# B&R Automation Studio project CControl_Gschneitner
Automation Studio 4.12.9.18 SP; technology packages: mapp 5.24.6

## Configuration 2_07

CPU 4PPC30.0702-21B, AutomationRuntime S4.93, Build 4.1.2, Safety 0.0, Vc V4.73.5

### Task classes (Cpu.sw)
```
Cyclic#1 (cycle 10000 us, tolerance 10000 us):
  eUhr <- Util.eUhr.prg
  UsbLink <- CSV.UsbLink.prg
Cyclic#2 (cycle 20000 us, tolerance 20000 us):
  hmiMain <- Visualisierung.hmiMain.prg
  System <- Util.System.prg
  StartStopp <- Steuerung.StartStopp.prg
  mappPara <- Util.mappPara.prg
Cyclic#3 (cycle 50000 us, tolerance 50000 us):
  io207 <- IO.io207.prg
  aktorenMap <- IO.aktorenMapping.prg
  boxenMappi <- IO.boxenMapping.prg
  Ablaufstrg <- Ablaufsteuerung.Ablaufstrg.prg
  Leistung <- Regelung.Leistung.prg
  Sitemanage <- Sitemanager.Sitemanager.prg
Cyclic#4 (cycle 100000 us, tolerance 100000 us):
  Nutzung <- Util.Nutzung.prg
  Alarm <- Alarmsystem.Alarm.prg
  Berechnung <- Berechnung.Berechnung.prg
Cyclic#5 (cycle 200000 us, tolerance 200000 us):
  Energiemes <- IO.Energiemessung.prg
  hmiConnect <- Visualisierung.hmiConnect.prg
Cyclic#6 (cycle 500000 us, tolerance 500000 us):
  CSV01_EXT <- CSV.CSV01_EXT.prg
  CSV01_PRG <- CSV.CSV01_PRG.prg
DataObjects: CSV01_CFG <- CSV.CSV01_CFG.dob
VcDataObjects: Visu <- Visualisierung.Visu.dob
Binaries: vccddbox, vccbtn, vcpdvnc, arialbd, vcmgr, vctcal, vcgclass, vcfile, vccnum, TCData, vcfntttf, vcpkat, vcdsloc, vcbclass, udbdef, FWRules, vcpd335x, vccstr, vccalarm, visvc, arial, Visu03, vccshape, vcalarm, vcpfppct, Visu01, vccdt, vcptelo, vcchspot, vcpk, vccbmp, vccpopup, vcshared, vcrt, vcnet, Visu02, vcctext, vcctrend, arsvcreg, vcclbox, vccbar, vcdsint, vcpdsw, vccovl, vccline, Config, sysconf, Role, User, ashwd, ashwac, iomap, arconfig, asfw
Libraries: operator, runtime, astime, AsIecCon, standard, sys_lib, AsBrStr, LascoMath, LascoReg, LascoTrock, LascoUtil, LaEntfV2, LascoBoxen, LoopConR, brsystem, asstring, FileIO, DataObj, AsARCfg, visapi, AsUSB, dvframe, IecCheck, MpBase, AsTCP, MpFile, MpRecipe, CControl, CSV, vcresman
```

### Hardware
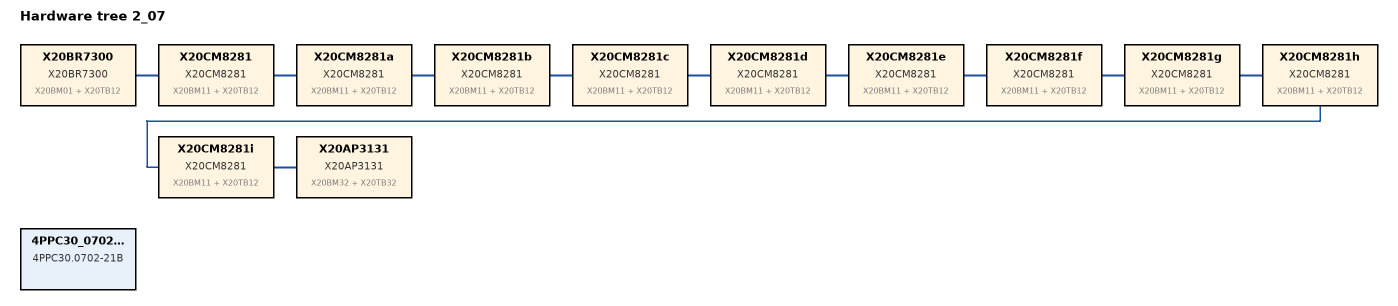
```
4PPC30_0702_21B : 4PPC30.0702-21B v1.1.4.0
  Connector IF3:
    ActivateDevice = 1
    Mode = Manual
    InternetAddress = 10.0.0.2
    SubnetMask = 255.255.255.0
    Vnc1
    VncVcObjectName1 = Visu
    VncKeyMappingFile1 = VC\PS2-Keyboard.dis
    VncMaxConnections1 = 5
    VncRefreshRate1 = 100
  Connector IF4:
    TerminatingResistor = 1
  ConfigurationID = CControl_2_07
  UserPartitionSize = 300
  RemanentGlobalPvSize = 7200
  EnableUsbRemoteInstall = 1
  TimerDeviceType = SWIOTIMER
  Cyclic1Duration = 10000
  Cyclic1Tolerance = 10000
  Cyclic2Duration = 20000
  Cyclic2Tolerance = 20000
  Cyclic3Duration = 50000
  Cyclic3Tolerance = 50000
  Cyclic4Duration = 100000
  Cyclic4Tolerance = 100000
  Cyclic5Duration = 200000
  Cyclic5Tolerance = 200000
  Cyclic6Duration = 500000
  Cyclic6Tolerance = 500000
  Cyclic7Duration = 1000000
  Cyclic7Tolerance = 1000000
  Cyclic8Duration = 10000
  Cyclic8Tolerance = 30000000
  FileDevice1
  FileDeviceName1 = CF
  FileDevicePath1 = F:\
  TimeZone = 140
  ActivateDaylightSavingTime = 1
  FtpUser1
  FtpUsername1 = lasco
  FtpUserPassword1 = KKiL+oKJhPTyxG5QFdiy6FHyy8yLLXpJAQupzJScLRk=
  FtpUserSalt1 = MRssQ874
  FTPAccessRight1 = 0
  FTPdevice1 = ALL
  VcObjectName = Visu
  KeyMappingFile = VC\4PPC30_0702_21B.dis
X20AP3131 : X20AP3131 v1.5.0.0  [SS1 -> X20TB32.SS; SL -> X20BM32.SL1]
  FunctionModel = CANIOBusController
  Supervision = off
  CurrentRatioA = 50
  CurrentRatioB = 50
  CurrentRatioC = 50
X20BM01 : X20BM01 v2.2.0.0
X20BM11 : X20BM11 v1.1.0.0  [X2X1 -> X20BM01.IF1]
X20BM11a : X20BM11 v1.1.0.0  [X2X1 -> X20BM11.X2X2]
X20BM11b : X20BM11 v1.1.0.0  [X2X1 -> X20BM11a.X2X2]
X20BM11c : X20BM11 v1.1.0.0  [X2X1 -> X20BM11b.X2X2]
X20BM11d : X20BM11 v1.1.0.0  [X2X1 -> X20BM11c.X2X2]
X20BM11e : X20BM11 v1.1.0.0  [X2X1 -> X20BM11d.X2X2]
X20BM11f : X20BM11 v1.1.0.0  [X2X1 -> X20BM11e.X2X2]
X20BM11g : X20BM11 v1.1.0.0  [X2X1 -> X20BM11f.X2X2]
X20BM11h : X20BM11 v1.1.0.0  [X2X1 -> X20BM11g.X2X2]
X20BM11i : X20BM11 v1.1.0.0  [X2X1 -> X20BM11h.X2X2]
X20BM32 : X20BM32 v1.1.0.0  [X2X1 -> X20BM11i.X2X2]
X20BR7300 : X20BR7300 v1.7.0.0  [CAN1 -> 4PPC30_0702_21B.IF4; SL -> X20BM01.SL1; SS1 -> X20TB12.SS]
  Supervision = off
X20CM8281 : X20CM8281 v1.4.0.0  [SS1 -> X20TB12a.SS; SL -> X20BM11.SL1]
  FunctionModel = CANIOBusController
  Supervision = off
  ChannelType01AI = 4 to 20mA
  LowerLimitAI = 0
  ChannelType01AO = 0 to 20mA
X20CM8281a : X20CM8281 v1.4.0.0  [SS1 -> X20TB12b.SS; SL -> X20BM11a.SL1]
  FunctionModel = CANIOBusController
  Supervision = off
  ChannelType01AI = 4 to 20mA
  LowerLimitAI = 0
  ChannelType01AO = 0 to 20mA
X20CM8281b : X20CM8281 v1.4.0.0  [SS1 -> X20TB12c.SS; SL -> X20BM11b.SL1]
  FunctionModel = CANIOBusController
  Supervision = off
  ChannelType01AI = 4 to 20mA
  LowerLimitAI = 0
  ChannelType01AO = 0 to 20mA
X20CM8281c : X20CM8281 v1.4.0.0  [SS1 -> X20TB12d.SS; SL -> X20BM11c.SL1]
  FunctionModel = CANIOBusController
  Supervision = off
  ChannelType01AI = 4 to 20mA
  LowerLimitAI = 0
X20CM8281d : X20CM8281 v1.4.0.0  [SS1 -> X20TB12e.SS; SL -> X20BM11d.SL1]
  FunctionModel = CANIOBusController
  Supervision = off
  ChannelType01AI = 4 to 20mA
  LowerLimitAI = 0
X20CM8281e : X20CM8281 v1.4.0.0  [SS1 -> X20TB12f.SS; SL -> X20BM11e.SL1]
  FunctionModel = CANIOBusController
  Supervision = off
  ChannelType01AI = 4 to 20mA
  LowerLimitAI = 0
X20CM8281f : X20CM8281 v1.4.0.0  [SS1 -> X20TB12g.SS; SL -> X20BM11f.SL1]
  FunctionModel = CANIOBusController
  Supervision = off
  ChannelType01AI = 4 to 20mA
  LowerLimitAI = 0
  ChannelType01AO = 0 to 20mA
X20CM8281g : X20CM8281 v1.4.0.0  [SS1 -> X20TB12h.SS; SL -> X20BM11g.SL1]
  FunctionModel = CANIOBusController
  Supervision = off
  ChannelType01AI = 4 to 20mA
  LowerLimitAI = 0
X20CM8281h : X20CM8281 v1.4.0.0  [SS1 -> X20TB12i.SS; SL -> X20BM11h.SL1]
  FunctionModel = CANIOBusController
  Supervision = off
X20CM8281i : X20CM8281 v1.4.0.0  [SS1 -> X20TB12j.SS; SL -> X20BM11i.SL1]
  FunctionModel = CANIOBusController
  Supervision = off
  ChannelType01AI = 4 to 20mA
X20TB12 : X20TB12 v1.0.0.0
X20TB12a : X20TB12 v1.0.0.0
X20TB12b : X20TB12 v1.0.0.0
X20TB12c : X20TB12 v1.0.0.0
X20TB12d : X20TB12 v1.0.0.0
X20TB12e : X20TB12 v1.0.0.0
X20TB12f : X20TB12 v1.0.0.0
X20TB12g : X20TB12 v1.0.0.0
X20TB12h : X20TB12 v1.0.0.0
X20TB12i : X20TB12 v1.0.0.0
X20TB12j : X20TB12 v1.0.0.0
X20TB32 : X20TB32 v1.0.0.1
```

### IoMap.iom - 4PPC30_0702_21B/IoMap.iom
```iecst
VAR_CONFIG
	::io207:brModul01.ModulOk AT %IX."X20BR7300".IF1.ST1.ModuleOk;
	::io207:cmModul02.ModulOk AT %IX."X20CM8281".ModuleOk;
	::io207:cmModul02.di01 AT %IX."X20CM8281".DigitalInput01;
	::io207:cmModul02.di02  AT %IX."X20CM8281".DigitalInput02;
	::io207:cmModul02.di03 AT %IX."X20CM8281".DigitalInput03;
	::io207:cmModul02.di04  AT %IX."X20CM8281".DigitalInput04;
	::io207:cmModul02.do01 AT %QX."X20CM8281".DigitalOutput01;
	::io207:cmModul02.do02 AT %QX."X20CM8281".DigitalOutput02;
	::io207:cmModul02.ai01 AT %IW."X20CM8281".AnalogInput01;
	::io207:cmModul02.ao01 AT %QW."X20CM8281".AnalogOutput01;
	::io207:cmModul02.StatusInput01 AT %IB."X20CM8281".StatusInput01;
	::io207:cmModul03.ModulOk AT %IX."X20CM8281a".ModuleOk;
	::io207:cmModul03.di01 AT %IX."X20CM8281a".DigitalInput01;
	::io207:cmModul03.di02  AT %IX."X20CM8281a".DigitalInput02;
	::io207:cmModul03.di03  AT %IX."X20CM8281a".DigitalInput03;
	::io207:cmModul03.di04  AT %IX."X20CM8281a".DigitalInput04;
	::io207:cmModul03.do01 AT %QX."X20CM8281a".DigitalOutput01;
	::io207:cmModul03.do02 AT %QX."X20CM8281a".DigitalOutput02;
	::io207:cmModul03.ai01 AT %IW."X20CM8281a".AnalogInput01;
	::io207:cmModul03.ao01 AT %QW."X20CM8281a".AnalogOutput01;
	::io207:cmModul03.StatusInput01 AT %IB."X20CM8281a".StatusInput01;
	::io207:cmModul04.ModulOk AT %IX."X20CM8281b".ModuleOk;
	::io207:cmModul04.di01 AT %IX."X20CM8281b".DigitalInput01;
	::io207:cmModul04.di02 AT %IX."X20CM8281b".DigitalInput02;
	::io207:cmModul04.di03 AT %IX."X20CM8281b".DigitalInput03;
	::io207:cmModul04.di04 AT %IX."X20CM8281b".DigitalInput04;
	::io207:cmModul04.do01 AT %QX."X20CM8281b".DigitalOutput01;
	::io207:cmModul04.do02 AT %QX."X20CM8281b".DigitalOutput02;
	::io207:cmModul04.ai01 AT %IW."X20CM8281b".AnalogInput01;
	::io207:cmModul04.ao01 AT %QW."X20CM8281b".AnalogOutput01;
	::io207:cmModul04.StatusInput01 AT %IB."X20CM8281b".StatusInput01;
	::io207:cmModul05.ModulOk AT %IX."X20CM8281c".ModuleOk;
	::io207:cmModul05.di01 AT %IX."X20CM8281c".DigitalInput01;
	::io207:cmModul05.di02 AT %IX."X20CM8281c".DigitalInput02;
	::io207:cmModul05.di03 AT %IX."X20CM8281c".DigitalInput03;
	::io207:cmModul05.di04 AT %IX."X20CM8281c".DigitalInput04;
	::io207:cmModul05.do01 AT %QX."X20CM8281c".DigitalOutput01;
	::io207:cmModul05.do02 AT %QX."X20CM8281c".DigitalOutput02;
	::io207:cmModul05.ai01 AT %IW."X20CM8281c".AnalogInput01;
	::io207:cmModul05.ao01 AT %QW."X20CM8281c".AnalogOutput01;
	::io207:cmModul05.StatusInput01 AT %IB."X20CM8281c".StatusInput01;
	::io207:cmModul06.ModulOk AT %IX."X20CM8281d".ModuleOk;
	::io207:cmModul06.di01 AT %IX."X20CM8281d".DigitalInput01;
	::io207:cmModul06.di02 AT %IX."X20CM8281d".DigitalInput02;
	::io207:cmModul06.di03 AT %IX."X20CM8281d".DigitalInput03;
	::io207:cmModul06.di04 AT %IX."X20CM8281d".DigitalInput04;
	::io207:cmModul06.do01 AT %QX."X20CM8281d".DigitalOutput01;
	::io207:cmModul06.do02 AT %QX."X20CM8281d".DigitalOutput02;
	::io207:cmModul06.ai01 AT %IW."X20CM8281d".AnalogInput01;
	::io207:cmModul06.ao01 AT %QW."X20CM8281d".AnalogOutput01;
	::io207:cmModul06.StatusInput01 AT %IB."X20CM8281d".StatusInput01;
	::io207:cmModul07.ModulOk AT %IX."X20CM8281e".ModuleOk;
	::io207:cmModul07.di01 AT %IX."X20CM8281e".DigitalInput01;
	::io207:cmModul07.di02 AT %IX."X20CM8281e".DigitalInput02;
	::io207:cmModul07.di03 AT %IX."X20CM8281e".DigitalInput03;
	::io207:cmModul07.di04 AT %IX."X20CM8281e".DigitalInput04;
	::io207:cmModul07.do01 AT %QX."X20CM8281e".DigitalOutput01;
	::io207:cmModul07.do02 AT %QX."X20CM8281e".DigitalOutput02;
	::io207:cmModul07.ai01 AT %IW."X20CM8281e".AnalogInput01;
	::io207:cmModul07.ao01 AT %QW."X20CM8281e".AnalogOutput01;
	::io207:cmModul07.StatusInput01 AT %IB."X20CM8281e".StatusInput01;
	::io207:cmModul08.ModulOk AT %IX."X20CM8281f".ModuleOk;
	::io207:cmModul08.di01 AT %IX."X20CM8281f".DigitalInput01;
	::io207:cmModul08.di02 AT %IX."X20CM8281f".DigitalInput02;
	::io207:cmModul08.di03 AT %IX."X20CM8281f".DigitalInput03;
	::io207:cmModul08.di04 AT %IX."X20CM8281f".DigitalInput04;
	::io207:cmModul08.do01 AT %QX."X20CM8281f".DigitalOutput01;
	::io207:cmModul08.do02 AT %QX."X20CM8281f".DigitalOutput02;
	::io207:cmModul08.ai01 AT %IW."X20CM8281f".AnalogInput01;
	::io207:cmModul08.ao01 AT %QW."X20CM8281f".AnalogOutput01;
	::io207:cmModul08.StatusInput01 AT %IB."X20CM8281f".StatusInput01;
	::io207:cmModul09.ModulOk AT %IX."X20CM8281g".ModuleOk;
	::io207:cmModul09.di01 AT %IX."X20CM8281g".DigitalInput01;
	::io207:cmModul09.di02 AT %IX."X20CM8281g".DigitalInput02;
	::io207:cmModul09.di03 AT %IX."X20CM8281g".DigitalInput03;
	::io207:cmModul09.di04 AT %IX."X20CM8281g".DigitalInput04;
	::io207:cmModul09.do01 AT %QX."X20CM8281g".DigitalOutput01;
	::io207:cmModul09.do02 AT %QX."X20CM8281g".DigitalOutput02;
	::io207:cmModul09.ai01 AT %IW."X20CM8281g".AnalogInput01;
	::io207:cmModul09.ao01 AT %QW."X20CM8281g".AnalogOutput01;
	::io207:cmModul09.StatusInput01 AT %IB."X20CM8281g".StatusInput01;
	::io207:cmModul10.ModulOk AT %IX."X20CM8281h".ModuleOk;
	::io207:cmModul10.di01 AT %IX."X20CM8281h".DigitalInput01;
	::io207:cmModul10.di02 AT %IX."X20CM8281h".DigitalInput02;
	::io207:cmModul10.di03 AT %IX."X20CM8281h".DigitalInput03;
	::io207:cmModul10.di04 AT %IX."X20CM8281h".DigitalInput04;
	::io207:cmModul10.do01 AT %QX."X20CM8281h".DigitalOutput01;
	::io207:cmModul10.do02 AT %QX."X20CM8281h".DigitalOutput02;
	::io207:cmModul10.ai01 AT %IW."X20CM8281h".AnalogInput01;
	::io207:cmModul10.ao01 AT %QW."X20CM8281h".AnalogOutput01;
	::io207:cmModul10.StatusInput01 AT %IB."X20CM8281h".StatusInput01;
	::io207:cmModul11.ModulOk AT %IX."X20CM8281i".ModuleOk;
	::io207:cmModul11.di01 AT %IX."X20CM8281i".DigitalInput01;
	::io207:cmModul11.di02 AT %IX."X20CM8281i".DigitalInput02;
	::io207:cmModul11.di03 AT %IX."X20CM8281i".DigitalInput03;
	::io207:cmModul11.di04 AT %IX."X20CM8281i".DigitalInput04;
	::io207:cmModul11.do01 AT %QX."X20CM8281i".DigitalOutput01;
	::io207:cmModul11.do02 AT %QX."X20CM8281i".DigitalOutput02;
	::io207:cmModul11.ai01 AT %IW."X20CM8281i".AnalogInput01;
	::io207:cmModul11.ao01 AT %QW."X20CM8281i".AnalogOutput01;
	::io207:cmModul11.StatusInput01 AT %IB."X20CM8281i".StatusInput01;
	::Energiemes:apModulEnergie.ModulOk AT %IX."X20AP3131".ModuleOk;
	::Energiemes:apModulEnergie.PmeanT AT %IW."X20AP3131".PmeanT;
	::Energiemes:apModulEnergie.QmeanT AT %IW."X20AP3131".QmeanT;
	::Energiemes:apModulEnergie.SmeanT AT %IW."X20AP3131".SmeanT;
	::Energiemes:apModulEnergie.PFmeanT AT %IW."X20AP3131".PFmeanT;
	::Energiemes:apModulEnergie.AenergyT AT %ID."X20AP3131".AenergyT;
	::Energiemes:apModulEnergie.RenergyT AT %ID."X20AP3131".RenergyT;
	::Energiemes:apModulEnergie.SAenergyT AT %ID."X20AP3131".SAenergyT;
	::Energiemes:apModulEnergie.RBClearEnergy AT %IX."X20AP3131".RBClearEnergy;
	::Energiemes:apModulEnergie.TrigDFT AT %QX."X20AP3131".TrigDFT;
	::Energiemes:apModulEnergie.EnabEnergy AT %QX."X20AP3131".EnabEnergy;
	::Energiemes:apModulEnergie.ClearEnergy AT %QX."X20AP3131".ClearEnergy;
	::Energiemes:apModulEnergie.ForceEnergy AT %QX."X20AP3131".ForceEnergy;
END_VAR
```

- Physical/2_07/4PPC30_0702_21B/PvMap.vvm: same as Physical/2_07/4PPC30_0702_21B/Cpu.per
### Config.mprecipexml - 4PPC30_0702_21B/mappServices/Config.mprecipexml
```
Element gMappRecipeLink (Type=mprecipexml)
```

## Configuration 3_04_Plus

CPU 4PPC30.043F-21B, AutomationRuntime S4.93, Build 4.1.2, Safety 0.0, Vc V4.73.5

### Task classes (Cpu.sw)
```
Cyclic#1 (cycle 10000 us, tolerance 10000 us):
  eUhr <- Util.eUhr.prg
  UsbLink <- CSV.UsbLink.prg
Cyclic#2 (cycle 20000 us, tolerance 20000 us):
  hmiMain <- Visualisierung.hmiMain.prg
  System <- Util.System.prg
  StartStopp <- Steuerung.StartStopp.prg
  mappPara <- Util.mappPara.prg
Cyclic#3 (cycle 50000 us, tolerance 50000 us):
  io304 <- IO.io304.prg  // IO-Konfiguration 3.04
  aktorenMap <- IO.aktorenMapping.prg
  boxenMappi <- IO.boxenMapping.prg
  Ablaufstrg <- Ablaufsteuerung.Ablaufstrg.prg
  Leistung <- Regelung.Leistung.prg
  Sitemanage <- Sitemanager.Sitemanager.prg
Cyclic#4 (cycle 100000 us, tolerance 100000 us):
  Nutzung <- Util.Nutzung.prg
  Berechnung <- Berechnung.Berechnung.prg
  Alarm <- Alarmsystem.Alarm.prg
Cyclic#5 (cycle 200000 us, tolerance 200000 us):
  hmiConnect <- Visualisierung.hmiConnect.prg
  Energiemes <- IO.Energiemessung.prg
Cyclic#6 (cycle 500000 us, tolerance 500000 us):
  CSV01_EXT <- CSV.CSV01_EXT.prg
  CSV01_PRG <- CSV.CSV01_PRG.prg
DataObjects: CSV01_CFG <- CSV.CSV01_CFG.dob
VcDataObjects: Visu4Z <- Visualisierung.Visu4Z.dob
Binaries: vccalarm, Visu4Z03, udbdef, vcrt, vccbar, vctcal, visvc, vccpopup, vcfile, vcgclass, vccstr, vcpdsw, vccshape, arial, vccbmp, vcmgr, vcshared, vcctrend, vcchspot, vcdsloc, Visu4Z01, vcctext, vccovl, vcfntttf, arialbd, vcpd335x, vccddbox, vcalarm, vcptelo, vccdt, vccline, vccbtn, Visu4Z02, vcbclass, vcdsint, vcpfppct, TCData, vcclbox, FWRules, vcpk, vccnum, arsvcreg, vcpdvnc, vcpkat, vcnet, sysconf, iomap, asfw, Role, ashwac, ashwd, User, arconfig, Config
Libraries: operator, runtime, astime, AsIecCon, standard, sys_lib, AsBrStr, LascoMath, LascoReg, LascoTrock, LascoUtil, LaEntfV2, LascoBoxen, LoopConR, brsystem, asstring, FileIO, DataObj, AsARCfg, visapi, AsUSB, dvframe, IecCheck, AsTCP, MpRecipe, MpBase, MpFile, CSV, CControl, vcresman
```

### Hardware
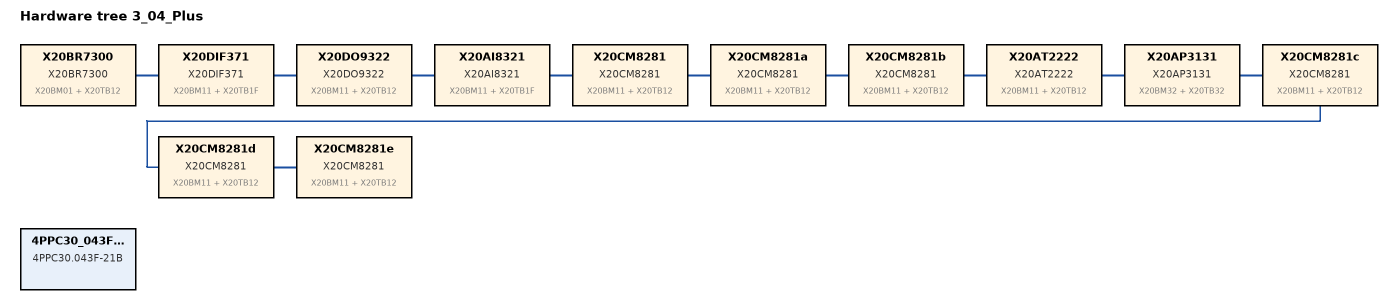
```
4PPC30_043F_21B : 4PPC30.043F-21B v1.1.3.0
  Connector IF3:
    ActivateDevice = 1
    Mode = Manual
    InternetAddress = 10.0.0.2
    SubnetMask = 255.255.255.0
    Vnc1
    VncVcObjectName1 = Visu4Z
    VncKeyMappingFile1 = VC\PS2-Keyboard.dis
    VncMaxConnections1 = 5
    VncRefreshRate1 = 100
  Connector IF4:
    TerminatingResistor = 1
  ConfigurationID = CControl304Plus
  UserPartitionSize = 200
  RemanentGlobalPvSize = 6000
  EnableUsbRemoteInstall = 1
  TimerDeviceType = SWIOTIMER
  Cyclic1Duration = 10000
  Cyclic1Tolerance = 10000
  Cyclic2Duration = 20000
  Cyclic2Tolerance = 20000
  Cyclic3Duration = 50000
  Cyclic3Tolerance = 50000
  Cyclic4Duration = 100000
  Cyclic4Tolerance = 100000
  Cyclic5Duration = 200000
  Cyclic5Tolerance = 200000
  Cyclic6Duration = 500000
  Cyclic6Tolerance = 500000
  Cyclic7Duration = 1000000
  Cyclic7Tolerance = 1000000
  Cyclic8Duration = 10000
  Cyclic8Tolerance = 30000000
  FileDevice1
  FileDeviceName1 = CF
  FileDevicePath1 = F:\
  FtpUser1
  FtpUsername1 = lasco
  FtpUserPassword1 = 97rNj208LBZIZPKyFvn5oul1tIa2LCmp2VBMYd1vER8=
  FtpUserSalt1 = M2zU6OPl
  FTPAccessRight1 = 0
  FTPdevice1 = ALL
  VcObjectName = Visu4Z
  RotationAngle = 180
  KeyMappingFile = VC\4PPC30_043F_21B.dis
X20AI8321 : X20AI8321 v1.5.0.0  [SS1 -> X20TB1F1.SS; SL -> X20BM11b.SL1]
  FunctionModel = CANIOBusController
  Supervision = off
  LowerLimit = 0
  ChannelType01 = 4 to 20mA
  ChannelType02 = 4 to 20mA
  ChannelType03 = 4 to 20mA
  ChannelType04 = 4 to 20mA
  ChannelType05 = 4 to 20mA
  ChannelType06 = 4 to 20mA
  ChannelType07 = 4 to 20mA
  ChannelType08 = 4 to 20mA
X20AP3131 : X20AP3131 v1.5.0.0  [SS1 -> X20TB32.SS; SL -> X20BM32.SL1]
  FunctionModel = CANIOBusController
  Supervision = off
  CurrentRatioA = 50
  CurrentRatioB = 50
  CurrentRatioC = 50
X20AT2222 : X20AT2222 v1.4.0.0  [SS1 -> X20TB12h.SS; SL -> X20BM11i.SL1]
  FunctionModel = CANIOBusController
  Supervision = off
X20BM01 : X20BM01 v2.2.0.0
X20BM11 : X20BM11 v1.1.0.0  [X2X1 -> X20BM01.IF1]
X20BM11a : X20BM11 v1.1.0.0  [X2X1 -> X20BM11.X2X2]
X20BM11b : X20BM11 v1.1.0.0  [X2X1 -> X20BM11a.X2X2]
X20BM11c : X20BM11 v1.1.0.0  [X2X1 -> X20BM11b.X2X2]
X20BM11d : X20BM11 v1.1.0.0  [X2X1 -> X20BM11c.X2X2]
X20BM11e : X20BM11 v1.1.0.0  [X2X1 -> X20BM11d.X2X2]
X20BM11f : X20BM11 v1.1.0.0  [X2X1 -> X20BM32.X2X2]
X20BM11g : X20BM11 v1.1.0.0  [X2X1 -> X20BM11f.X2X2]
X20BM11h : X20BM11 v1.1.0.0  [X2X1 -> X20BM11g.X2X2]
X20BM11i : X20BM11 v1.1.0.0  [X2X1 -> X20BM11e.X2X2]
X20BM32 : X20BM32 v1.1.0.0  [X2X1 -> X20BM11i.X2X2]
X20BR7300 : X20BR7300 v1.7.0.0  [CAN1 -> 4PPC30_043F_21B.IF4; SL -> X20BM01.SL1; SS1 -> X20TB12.SS]
  Supervision = off
X20CM8281 : X20CM8281 v1.4.0.0  [SS1 -> X20TB12b.SS; SL -> X20BM11c.SL1]
  FunctionModel = CANIOBusController
  Supervision = off
  ChannelType01AO = 0 to 20mA
X20CM8281a : X20CM8281 v1.4.0.0  [SS1 -> X20TB12c.SS; SL -> X20BM11d.SL1]
  FunctionModel = CANIOBusController
  Supervision = off
  ChannelType01AI = 4 to 20mA
  LowerLimitAI = 0
  ChannelType01AO = 0 to 20mA
X20CM8281b : X20CM8281 v1.4.0.0  [SS1 -> X20TB12d.SS; SL -> X20BM11e.SL1]
  FunctionModel = CANIOBusController
  Supervision = off
  ChannelType01AI = 4 to 20mA
  LowerLimitAI = 0
X20CM8281c : X20CM8281 v1.4.0.0  [SS1 -> X20TB12e.SS; SL -> X20BM11f.SL1]
  FunctionModel = CANIOBusController
  Supervision = off
  ChannelType01AI = 4 to 20mA
  LowerLimitAI = 0
  ChannelType01AO = 0 to 20mA
X20CM8281d : X20CM8281 v1.4.0.0  [SS1 -> X20TB12f.SS; SL -> X20BM11g.SL1]
  FunctionModel = CANIOBusController
  Supervision = off
  ChannelType01AI = 4 to 20mA
  LowerLimitAI = 0
  ChannelType01AO = 0 to 20mA
X20CM8281e : X20CM8281 v1.4.0.0  [SS1 -> X20TB12g.SS; SL -> X20BM11h.SL1]
  FunctionModel = CANIOBusController
  Supervision = off
  ChannelType01AI = 4 to 20mA
X20DIF371 : X20DIF371 v1.3.0.0  [SS1 -> X20TB1F.SS; SL -> X20BM11.SL1]
  FunctionModel = CANIOBusController
  Supervision = off
X20DO9322 : X20DO9322 v1.7.0.0  [SS1 -> X20TB12a.SS; SL -> X20BM11a.SL1]
  FunctionModel = CANIOBusController
  Supervision = off
X20TB12 : X20TB12 v1.0.0.0
X20TB12a : X20TB12 v1.0.0.0
X20TB12b : X20TB12 v1.0.0.0
X20TB12c : X20TB12 v1.0.0.0
X20TB12d : X20TB12 v1.0.0.0
X20TB12e : X20TB12 v1.0.0.0
X20TB12f : X20TB12 v1.0.0.0
X20TB12g : X20TB12 v1.0.0.0
X20TB12h : X20TB12 v1.0.0.0
X20TB1F : X20TB1F v1.0.0.0
X20TB1F1 : X20TB1F v1.0.0.0
X20TB32 : X20TB32 v1.0.0.1
```

- Physical/3_04_Plus/4PPC30_043F_21B/Cpu.per: same as Physical/2_07/4PPC30_0702_21B/Cpu.per
### IoMap.iom - 4PPC30_043F_21B/IoMap.iom
```iecst
VAR_CONFIG
	::io304:brModul01.ModulOk AT %IX."X20BR7300".IF1.ST1.ModuleOk;
	::io304:diModul02.ModulOk AT %IX."X20DIF371".ModuleOk;
	::io304:diModul02.di01 AT %IX."X20DIF371".DigitalInput01;
	::io304:diModul02.di02 AT %IX."X20DIF371".DigitalInput02;
	::io304:diModul02.di03 AT %IX."X20DIF371".DigitalInput03;
	::io304:diModul02.di04 AT %IX."X20DIF371".DigitalInput04;
	::io304:diModul02.di05 AT %IX."X20DIF371".DigitalInput05;
	::io304:diModul02.di06 AT %IX."X20DIF371".DigitalInput06;
	::io304:diModul02.di07 AT %IX."X20DIF371".DigitalInput07;
	::io304:diModul02.di08 AT %IX."X20DIF371".DigitalInput08;
	::io304:diModul02.di09 AT %IX."X20DIF371".DigitalInput09;
	::io304:diModul02.di10 AT %IX."X20DIF371".DigitalInput10;
	::io304:diModul02.di11 AT %IX."X20DIF371".DigitalInput11;
	::io304:diModul02.di12 AT %IX."X20DIF371".DigitalInput12;
	::io304:diModul02.di13 AT %IX."X20DIF371".DigitalInput13;
	::io304:diModul02.di14 AT %IX."X20DIF371".DigitalInput14;
	::io304:diModul02.di15 AT %IX."X20DIF371".DigitalInput15;
	::io304:diModul02.di16 AT %IX."X20DIF371".DigitalInput16;
	::io304:doModul03.ModulOk AT %IX."X20DO9322".ModuleOk;
	::io304:doModul03.do01 AT %QX."X20DO9322".DigitalOutput01;
	::io304:doModul03.do02 AT %QX."X20DO9322".DigitalOutput02;
	::io304:doModul03.do03 AT %QX."X20DO9322".DigitalOutput03;
	::io304:doModul03.do04 AT %QX."X20DO9322".DigitalOutput04;
	::io304:doModul03.do05 AT %QX."X20DO9322".DigitalOutput05;
	::io304:doModul03.do06 AT %QX."X20DO9322".DigitalOutput06;
	::io304:doModul03.do07 AT %QX."X20DO9322".DigitalOutput07;
	::io304:doModul03.do08 AT %QX."X20DO9322".DigitalOutput08;
	::io304:doModul03.do09 AT %QX."X20DO9322".DigitalOutput09;
	::io304:doModul03.do10 AT %QX."X20DO9322".DigitalOutput10;
	::io304:doModul03.do11 AT %QX."X20DO9322".DigitalOutput11;
	::io304:doModul03.do12 AT %QX."X20DO9322".DigitalOutput12;
	::io304:aiModul04.ModulOk AT %IX."X20AI8321".ModuleOk;
	::io304:aiModul04.ai01 AT %IW."X20AI8321".AnalogInput01;
	::io304:aiModul04.ai02 AT %IW."X20AI8321".AnalogInput02;
	::io304:aiModul04.ai03 AT %IW."X20AI8321".AnalogInput03;
	::io304:aiModul04.ai04 AT %IW."X20AI8321".AnalogInput04;
	::io304:aiModul04.ai05 AT %IW."X20AI8321".AnalogInput05;
	::io304:aiModul04.ai06 AT %IW."X20AI8321".AnalogInput06;
	::io304:aiModul04.ai07 AT %IW."X20AI8321".AnalogInput07;
	::io304:aiModul04.ai08 AT %IW."X20AI8321".AnalogInput08;
	::io304:aiModul04.StatusInput01 AT %IB."X20AI8321".StatusInput01;
	::io304:aiModul04.StatusInput02 AT %IB."X20AI8321".StatusInput02;
	::io304:cmModul05.ModulOk AT %IX."X20CM8281".ModuleOk;
	::io304:cmModul05.di01 AT %IX."X20CM8281".DigitalInput01;
	::io304:cmModul05.di02 AT %IX."X20CM8281".DigitalInput02;
	::io304:cmModul05.di03 AT %IX."X20CM8281".DigitalInput03;
	::io304:cmModul05.di04 AT %IX."X20CM8281".DigitalInput04;
	::io304:cmModul05.do01 AT %QX."X20CM8281".DigitalOutput01;
	::io304:cmModul05.do02 AT %QX."X20CM8281".DigitalOutput02;
	::io304:cmModul05.ai01 AT %IW."X20CM8281".AnalogInput01;
	::io304:cmModul05.ao01 AT %QW."X20CM8281".AnalogOutput01;
	::io304:cmModul05.StatusInput01 AT %IB."X20CM8281".StatusInput01;
	::io304:cmModul06.ModulOk AT %IX."X20CM8281a".ModuleOk;
	::io304:cmModul06.di01 AT %IX."X20CM8281a".DigitalInput01;
	::io304:cmModul06.di02 AT %IX."X20CM8281a".DigitalInput02;
	::io304:cmModul06.di03 AT %IX."X20CM8281a".DigitalInput03;
	::io304:cmModul06.di04 AT %IX."X20CM8281a".DigitalInput04;
	::io304:cmModul06.do01 AT %QX."X20CM8281a".DigitalOutput01;
	::io304:cmModul06.do02 AT %QX."X20CM8281a".DigitalOutput02;
	::io304:cmModul06.ai01 AT %IW."X20CM8281a".AnalogInput01;
	::io304:cmModul06.ao01 AT %QW."X20CM8281a".AnalogOutput01;
	::io304:cmModul06.StatusInput01 AT %IB."X20CM8281a".StatusInput01;
	::io304:cmModul07.ModulOk AT %IX."X20CM8281b".ModuleOk;
	::io304:cmModul07.di01 AT %IX."X20CM8281b".DigitalInput01;
	::io304:cmModul07.di02 AT %IX."X20CM8281b".DigitalInput02;
	::io304:cmModul07.di03 AT %IX."X20CM8281b".DigitalInput03;
	::io304:cmModul07.di04 AT %IX."X20CM8281b".DigitalInput04;
	::io304:cmModul07.do01 AT %QX."X20CM8281b".DigitalOutput01;
	::io304:cmModul07.do02 AT %QX."X20CM8281b".DigitalOutput02;
	::io304:cmModul07.ai01 AT %IW."X20CM8281b".AnalogInput01;
	::io304:cmModul07.ao01 AT %QW."X20CM8281b".AnalogOutput01;
	::io304:cmModul07.StatusInput01 AT %IB."X20CM8281b".StatusInput01;
	::Energiemes:apModulEnergie.ModulOk AT %IX."X20AP3131".ModuleOk;
	::Energiemes:apModulEnergie.PmeanT AT %IW."X20AP3131".PmeanT;
	::Energiemes:apModulEnergie.QmeanT AT %IW."X20AP3131".QmeanT;
	::Energiemes:apModulEnergie.SmeanT AT %IW."X20AP3131".SmeanT;
	::Energiemes:apModulEnergie.PFmeanT AT %IW."X20AP3131".PFmeanT;
	::Energiemes:apModulEnergie.AenergyT AT %ID."X20AP3131".AenergyT;
	::Energiemes:apModulEnergie.RenergyT AT %ID."X20AP3131".RenergyT;
	::Energiemes:apModulEnergie.SAenergyT AT %ID."X20AP3131".SAenergyT;
	::Energiemes:apModulEnergie.RBClearEnergy AT %IX."X20AP3131".RBClearEnergy;
	::Energiemes:apModulEnergie.TrigDFT AT %QX."X20AP3131".TrigDFT;
	::Energiemes:apModulEnergie.EnabEnergy AT %QX."X20AP3131".EnabEnergy;
	::Energiemes:apModulEnergie.ClearEnergy AT %QX."X20AP3131".ClearEnergy;
	::Energiemes:apModulEnergie.ForceEnergy AT %QX."X20AP3131".ForceEnergy;
	::io304:cmModul10.ModulOk AT %IX."X20CM8281c".ModuleOk;
	::io304:cmModul10.di01 AT %IX."X20CM8281c".DigitalInput01;
	::io304:cmModul10.di02 AT %IX."X20CM8281c".DigitalInput02;
	::io304:cmModul10.di03 AT %IX."X20CM8281c".DigitalInput03;
	::io304:cmModul10.di04 AT %IX."X20CM8281c".DigitalInput04;
	::io304:cmModul10.do01 AT %QX."X20CM8281c".DigitalOutput01;
	::io304:cmModul10.do02 AT %QX."X20CM8281c".DigitalOutput02;
	::io304:cmModul10.ai01 AT %IW."X20CM8281c".AnalogInput01;
	::io304:cmModul10.ao01 AT %QW."X20CM8281c".AnalogOutput01;
	::io304:cmModul10.StatusInput01 AT %IB."X20CM8281c".StatusInput01;
	::io304:cmModul11.ModulOk AT %IX."X20CM8281d".ModuleOk;
	::io304:cmModul11.di01 AT %IX."X20CM8281d".DigitalInput01;
	::io304:cmModul11.di02 AT %IX."X20CM8281d".DigitalInput02;
	::io304:cmModul11.di03 AT %IX."X20CM8281d".DigitalInput03;
	::io304:cmModul11.di04 AT %IX."X20CM8281d".DigitalInput04;
	::io304:cmModul11.do01 AT %QX."X20CM8281d".DigitalOutput01;
	::io304:cmModul11.do02 AT %QX."X20CM8281d".DigitalOutput02;
	::io304:cmModul11.ai01 AT %IW."X20CM8281d".AnalogInput01;
	::io304:cmModul11.ao01 AT %QW."X20CM8281d".AnalogOutput01;
	::io304:cmModul11.StatusInput01 AT %IB."X20CM8281d".StatusInput01;
	::io304:cmModul12.ModulOk AT %IX."X20CM8281e".ModuleOk;
	::io304:cmModul12.di01 AT %IX."X20CM8281e".DigitalInput01;
	::io304:cmModul12.di02 AT %IX."X20CM8281e".DigitalInput02;
	::io304:cmModul12.di03 AT %IX."X20CM8281e".DigitalInput03;
	::io304:cmModul12.di04 AT %IX."X20CM8281e".DigitalInput04;
	::io304:cmModul12.do01 AT %QX."X20CM8281e".DigitalOutput01;
	::io304:cmModul12.do02 AT %QX."X20CM8281e".DigitalOutput02;
	::io304:cmModul12.ai01 AT %IW."X20CM8281e".AnalogInput01;
	::io304:cmModul12.ao01 AT %QW."X20CM8281e".AnalogOutput01;
	::io304:cmModul12.StatusInput01 AT %IB."X20CM8281e".StatusInput01;
	::io304:atModul08.ModulOk AT %IX."X20AT2222".ModuleOk;
	::io304:atModul08.at01 AT %IW."X20AT2222".Temperature01;
	::io304:atModul08.at02 AT %IW."X20AT2222".Temperature02;
	::io304:atModul08.StatusInput01 AT %IB."X20AT2222".StatusInput01;
END_VAR
```

- Physical/3_04_Plus/4PPC30_043F_21B/PvMap.vvm: same as Physical/2_07/4PPC30_0702_21B/Cpu.per
### Config.mprecipexml - 4PPC30_043F_21B/mappServices/Config.mprecipexml
```
Element gMappRecipeLink (Type=mprecipexml)
  mapp.Recipe.Xml:
    PassPhrase = 
```

## Configuration 3_07

CPU 4PPC30.0702-21B, AutomationRuntime S4.93, Build 4.1.2, Vc V4.73.5

### Task classes (Cpu.sw)
```
Cyclic#1 (cycle 10000 us, tolerance 10000 us):
  eUhr <- Util.eUhr.prg
  UsbLink <- CSV.UsbLink.prg
Cyclic#2 (cycle 20000 us, tolerance 20000 us):
  hmiMain <- Visualisierung.hmiMain.prg
  System <- Util.System.prg
  StartStopp <- Steuerung.StartStopp.prg
  mappPara <- Util.mappPara.prg
Cyclic#3 (cycle 50000 us, tolerance 50000 us):
  io307 <- IO.io307.prg
  aktorenMap <- IO.aktorenMapping.prg
  boxenMappi <- IO.boxenMapping.prg
  Ablaufstrg <- Ablaufsteuerung.Ablaufstrg.prg
  Leistung <- Regelung.Leistung.prg
  Sitemanage <- Sitemanager.Sitemanager.prg
Cyclic#4 (cycle 100000 us, tolerance 100000 us):
  Nutzung <- Util.Nutzung.prg
  Berechnung <- Berechnung.Berechnung.prg
  Alarm <- Alarmsystem.Alarm.prg
Cyclic#5 (cycle 200000 us, tolerance 200000 us):
  Energiemes <- IO.Energiemessung.prg
  hmiConnect <- Visualisierung.hmiConnect.prg
Cyclic#6 (cycle 500000 us, tolerance 500000 us):
  CSV01_EXT <- CSV.CSV01_EXT.prg
  CSV01_PRG <- CSV.CSV01_PRG.prg
DataObjects: CSV01_CFG <- CSV.CSV01_CFG.dob
VcDataObjects: Visu <- Visualisierung.Visu.dob
Binaries: vccddbox, vccbtn, vcpdvnc, arialbd, vcmgr, vctcal, vcgclass, vcfile, vccnum, TCData, vcfntttf, vcpkat, vcdsloc, vcbclass, udbdef, FWRules, vcpd335x, vccstr, vccalarm, visvc, arial, Visu03, vccshape, vcalarm, vcpfppct, Visu01, vccdt, vcptelo, vcchspot, vcpk, vccbmp, vccpopup, vcshared, vcrt, vcnet, Visu02, vcctext, vcctrend, arsvcreg, vcclbox, vccbar, vcdsint, vcpdsw, vccovl, vccline, Config, sysconf, Role, User, ashwd, ashwac, iomap, arconfig, asfw
Libraries: MpRecipe, MpBase, sys_lib, runtime, operator, astime, AsIecCon, standard, AsBrStr, LascoMath, LascoReg, LascoTrock, LascoUtil, LaEntfV2, LascoBoxen, LoopConR, brsystem, asstring, FileIO, DataObj, AsARCfg, visapi, AsUSB, dvframe, IecCheck, AsTCP, CSV, MpFile, CControl, vcresman
```

### Hardware
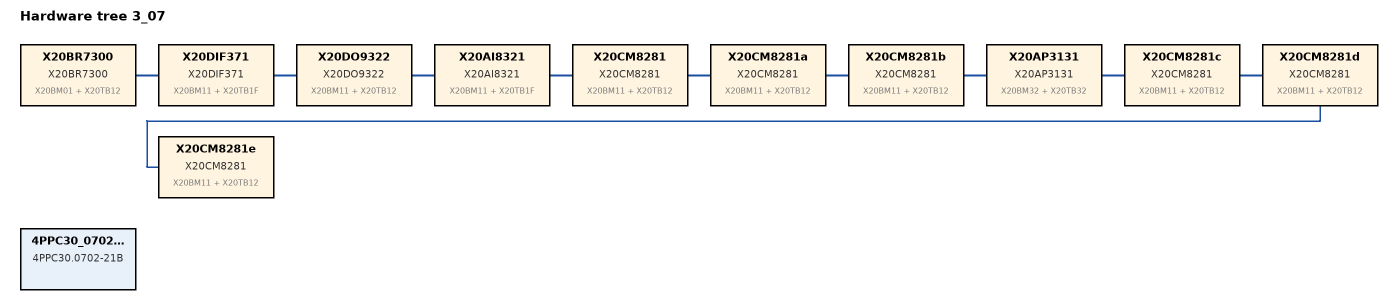
```
4PPC30_0702_21B : 4PPC30.0702-21B v1.1.4.0
  Connector IF3:
    ActivateDevice = 1
    Mode = Manual
    InternetAddress = 10.0.0.2
    SubnetMask = 255.255.255.0
    Vnc1
    VncVcObjectName1 = Visu
    VncKeyMappingFile1 = VC\PS2-Keyboard.dis
    VncMaxConnections1 = 5
    VncRefreshRate1 = 100
  Connector IF4:
    TerminatingResistor = 1
  ConfigurationID = CControl307_3_07
  UserPartitionSize = 300
  RemanentGlobalPvSize = 6000
  EnableUsbRemoteInstall = 1
  TimerDeviceType = SWIOTIMER
  Cyclic1Duration = 10000
  Cyclic1Tolerance = 10000
  Cyclic2Duration = 20000
  Cyclic2Tolerance = 20000
  Cyclic3Duration = 50000
  Cyclic3Tolerance = 50000
  Cyclic4Duration = 100000
  Cyclic4Tolerance = 100000
  Cyclic5Duration = 200000
  Cyclic5Tolerance = 200000
  Cyclic6Duration = 500000
  Cyclic6Tolerance = 500000
  Cyclic7Duration = 1000000
  Cyclic7Tolerance = 1000000
  Cyclic8Duration = 10000
  Cyclic8Tolerance = 30000000
  FileDevice1
  FileDeviceName1 = CF
  FileDevicePath1 = F:\
  TimeZone = 140
  ActivateDaylightSavingTime = 1
  FtpUser1
  FtpUsername1 = lasco
  FtpUserPassword1 = uMnLbGoaEITaZu0aep9FGD4ICFvOFtVGX1HqFSJwghw=
  FtpUserSalt1 = Q/JeTVjw
  FTPAccessRight1 = 0
  FTPdevice1 = ALL
  VcObjectName = Visu
  KeyMappingFile = VC\4PPC30_0702_21B.dis
X20AI8321 : X20AI8321 v1.5.0.0  [SS1 -> X20TB1F1.SS; SL -> X20BM11b.SL1]
  FunctionModel = CANIOBusController
  Supervision = off
  LowerLimit = 0
  ChannelType01 = 4 to 20mA
  ChannelType02 = 4 to 20mA
  ChannelType03 = 4 to 20mA
  ChannelType04 = 4 to 20mA
  ChannelType05 = 4 to 20mA
  ChannelType06 = 4 to 20mA
  ChannelType07 = 4 to 20mA
  ChannelType08 = 4 to 20mA
X20AP3131 : X20AP3131 v1.5.0.0  [SS1 -> X20TB32.SS; SL -> X20BM32.SL1]
  FunctionModel = CANIOBusController
  Supervision = off
  CurrentRatioA = 50
  CurrentRatioB = 50
  CurrentRatioC = 50
X20BM01 : X20BM01 v2.2.0.0
X20BM11 : X20BM11 v1.1.0.0  [X2X1 -> X20BM01.IF1]
X20BM11a : X20BM11 v1.1.0.0  [X2X1 -> X20BM11.X2X2]
X20BM11b : X20BM11 v1.1.0.0  [X2X1 -> X20BM11a.X2X2]
X20BM11c : X20BM11 v1.1.0.0  [X2X1 -> X20BM11b.X2X2]
X20BM11d : X20BM11 v1.1.0.0  [X2X1 -> X20BM11c.X2X2]
X20BM11e : X20BM11 v1.1.0.0  [X2X1 -> X20BM11d.X2X2]
X20BM11f : X20BM11 v1.1.0.0  [X2X1 -> X20BM11h.X2X2]
X20BM11g : X20BM11 v1.1.0.0  [X2X1 -> X20BM32.X2X2]
X20BM11h : X20BM11 v1.1.0.0  [X2X1 -> X20BM11g.X2X2]
X20BM32 : X20BM32 v1.1.0.0  [X2X1 -> X20BM11e.X2X2]
X20BR7300 : X20BR7300 v1.7.0.0  [CAN1 -> 4PPC30_0702_21B.IF4; SL -> X20BM01.SL1; SS1 -> X20TB12.SS]
  Supervision = off
X20CM8281 : X20CM8281 v1.4.0.0  [SS1 -> X20TB12b.SS; SL -> X20BM11c.SL1]
  FunctionModel = CANIOBusController
  Supervision = off
  ChannelType01AO = 0 to 20mA
X20CM8281a : X20CM8281 v1.4.0.0  [SS1 -> X20TB12c.SS; SL -> X20BM11d.SL1]
  FunctionModel = CANIOBusController
  Supervision = off
  ChannelType01AI = 4 to 20mA
  LowerLimitAI = 0
  ChannelType01AO = 0 to 20mA
X20CM8281b : X20CM8281 v1.4.0.0  [SS1 -> X20TB12d.SS; SL -> X20BM11e.SL1]
  FunctionModel = CANIOBusController
  Supervision = off
  ChannelType01AI = 4 to 20mA
  LowerLimitAI = 0
X20CM8281c : X20CM8281 v1.4.0.0  [SS1 -> X20TB12f.SS; SL -> X20BM11g.SL1]
  FunctionModel = CANIOBusController
  Supervision = off
  ChannelType01AI = 4 to 20mA
  LowerLimitAI = 0
  ChannelType01AO = 0 to 20mA
X20CM8281d : X20CM8281 v1.4.0.0  [SS1 -> X20TB12g.SS; SL -> X20BM11h.SL1]
  FunctionModel = CANIOBusController
  Supervision = off
  ChannelType01AI = 4 to 20mA
  LowerLimitAI = 0
  ChannelType01AO = 0 to 20mA
X20CM8281e : X20CM8281 v1.4.0.0  [SS1 -> X20TB12e.SS; SL -> X20BM11f.SL1]
  FunctionModel = CANIOBusController
  Supervision = off
  ChannelType01AI = 4 to 20mA
X20DIF371 : X20DIF371 v1.3.0.0  [SS1 -> X20TB1F.SS; SL -> X20BM11.SL1]
  FunctionModel = CANIOBusController
  Supervision = off
X20DO9322 : X20DO9322 v1.7.0.0  [SS1 -> X20TB12a.SS; SL -> X20BM11a.SL1]
  FunctionModel = CANIOBusController
  Supervision = off
X20TB12 : X20TB12 v1.0.0.0
X20TB12a : X20TB12 v1.0.0.0
X20TB12b : X20TB12 v1.0.0.0
X20TB12c : X20TB12 v1.0.0.0
X20TB12d : X20TB12 v1.0.0.0
X20TB12e : X20TB12 v1.0.0.0
X20TB12f : X20TB12 v1.0.0.0
X20TB12g : X20TB12 v1.0.0.0
X20TB1F : X20TB1F v1.0.0.0
X20TB1F1 : X20TB1F v1.0.0.0
X20TB32 : X20TB32 v1.0.0.1
```

- Physical/3_07/4PPC30_0702_21B/Cpu.per: same as Physical/2_07/4PPC30_0702_21B/Cpu.per
### IoMap.iom - 4PPC30_0702_21B/IoMap.iom
```iecst
VAR_CONFIG
	::io307:diModul02.di01 AT %IX."X20DIF371".DigitalInput01;
	::io307:diModul02.di02 AT %IX."X20DIF371".DigitalInput02;
	::io307:diModul02.di03 AT %IX."X20DIF371".DigitalInput03;
	::io307:diModul02.di04 AT %IX."X20DIF371".DigitalInput04;
	::io307:diModul02.di05 AT %IX."X20DIF371".DigitalInput05;
	::io307:diModul02.di06 AT %IX."X20DIF371".DigitalInput06;
	::io307:diModul02.di07 AT %IX."X20DIF371".DigitalInput07;
	::io307:diModul02.di08 AT %IX."X20DIF371".DigitalInput08;
	::io307:diModul02.di09 AT %IX."X20DIF371".DigitalInput09;
	::io307:diModul02.di10 AT %IX."X20DIF371".DigitalInput10;
	::io307:diModul02.di11 AT %IX."X20DIF371".DigitalInput11;
	::io307:diModul02.di12 AT %IX."X20DIF371".DigitalInput12;
	::io307:diModul02.di13 AT %IX."X20DIF371".DigitalInput13;
	::io307:diModul02.di14 AT %IX."X20DIF371".DigitalInput14;
	::io307:diModul02.di15 AT %IX."X20DIF371".DigitalInput15;
	::io307:diModul02.di16 AT %IX."X20DIF371".DigitalInput16;
	::io307:doModul03.do01 AT %QX."X20DO9322".DigitalOutput01;
	::io307:doModul03.do02 AT %QX."X20DO9322".DigitalOutput02;
	::io307:doModul03.do03 AT %QX."X20DO9322".DigitalOutput03;
	::io307:doModul03.do04 AT %QX."X20DO9322".DigitalOutput04;
	::io307:doModul03.do05 AT %QX."X20DO9322".DigitalOutput05;
	::io307:doModul03.do06 AT %QX."X20DO9322".DigitalOutput06;
	::io307:doModul03.do07 AT %QX."X20DO9322".DigitalOutput07;
	::io307:doModul03.do08 AT %QX."X20DO9322".DigitalOutput08;
	::io307:doModul03.do09 AT %QX."X20DO9322".DigitalOutput09;
	::io307:doModul03.do10 AT %QX."X20DO9322".DigitalOutput10;
	::io307:doModul03.do11 AT %QX."X20DO9322".DigitalOutput11;
	::io307:doModul03.do12 AT %QX."X20DO9322".DigitalOutput12;
	::io307:aiModul04.ai01 AT %IW."X20AI8321".AnalogInput01;
	::io307:aiModul04.ai02 AT %IW."X20AI8321".AnalogInput02;
	::io307:aiModul04.ai03 AT %IW."X20AI8321".AnalogInput03;
	::io307:aiModul04.ai04 AT %IW."X20AI8321".AnalogInput04;
	::io307:aiModul04.ai05 AT %IW."X20AI8321".AnalogInput05;
	::io307:aiModul04.ai06 AT %IW."X20AI8321".AnalogInput06;
	::io307:aiModul04.ai07 AT %IW."X20AI8321".AnalogInput07;
	::io307:aiModul04.ai08 AT %IW."X20AI8321".AnalogInput08;
	::io307:aiModul04.StatusInput01 AT %IB."X20AI8321".StatusInput01;
	::io307:aiModul04.StatusInput02 AT %IB."X20AI8321".StatusInput02;
	::io307:cmModul05.di01 AT %IX."X20CM8281".DigitalInput01;
	::io307:cmModul05.di02 AT %IX."X20CM8281".DigitalInput02;
	::io307:cmModul05.di03 AT %IX."X20CM8281".DigitalInput03;
	::io307:cmModul05.di04 AT %IX."X20CM8281".DigitalInput04;
	::io307:cmModul05.do01 AT %QX."X20CM8281".DigitalOutput01;
	::io307:cmModul05.do02 AT %QX."X20CM8281".DigitalOutput02;
	::io307:cmModul05.ai01 AT %IW."X20CM8281".AnalogInput01;
	::io307:cmModul05.ao01 AT %QW."X20CM8281".AnalogOutput01;
	::io307:cmModul05.StatusInput01 AT %IB."X20CM8281".StatusInput01;
	::io307:cmModul06.di01 AT %IX."X20CM8281a".DigitalInput01;
	::io307:cmModul06.di02 AT %IX."X20CM8281a".DigitalInput02;
	::io307:cmModul06.di03 AT %IX."X20CM8281a".DigitalInput03;
	::io307:cmModul06.di04 AT %IX."X20CM8281a".DigitalInput04;
	::io307:cmModul06.do01 AT %QX."X20CM8281a".DigitalOutput01;
	::io307:cmModul06.do02 AT %QX."X20CM8281a".DigitalOutput02;
	::io307:cmModul06.ai01 AT %IW."X20CM8281a".AnalogInput01;
	::io307:cmModul06.ao01 AT %QW."X20CM8281a".AnalogOutput01;
	::io307:cmModul06.StatusInput01 AT %IB."X20CM8281a".StatusInput01;
	::io307:cmModul07.di01 AT %IX."X20CM8281b".DigitalInput01;
	::io307:cmModul07.di02 AT %IX."X20CM8281b".DigitalInput02;
	::io307:cmModul07.di03 AT %IX."X20CM8281b".DigitalInput03;
	::io307:cmModul07.di04 AT %IX."X20CM8281b".DigitalInput04;
	::io307:cmModul07.do01 AT %QX."X20CM8281b".DigitalOutput01;
	::io307:cmModul07.do02 AT %QX."X20CM8281b".DigitalOutput02;
	::io307:cmModul07.ai01 AT %IW."X20CM8281b".AnalogInput01;
	::io307:cmModul07.ao01 AT %QW."X20CM8281b".AnalogOutput01;
	::io307:cmModul07.StatusInput01 AT %IB."X20CM8281b".StatusInput01;
	::Energiemes:apModulEnergie.PmeanT AT %IW."X20AP3131".PmeanT;
	::Energiemes:apModulEnergie.QmeanT AT %IW."X20AP3131".QmeanT;
	::Energiemes:apModulEnergie.SmeanT AT %IW."X20AP3131".SmeanT;
	::Energiemes:apModulEnergie.PFmeanT AT %IW."X20AP3131".PFmeanT;
	::Energiemes:apModulEnergie.AenergyT AT %ID."X20AP3131".AenergyT;
	::Energiemes:apModulEnergie.RenergyT AT %ID."X20AP3131".RenergyT;
	::Energiemes:apModulEnergie.SAenergyT AT %ID."X20AP3131".SAenergyT;
	::Energiemes:apModulEnergie.RBClearEnergy AT %IX."X20AP3131".RBClearEnergy;
	::Energiemes:apModulEnergie.TrigDFT AT %QX."X20AP3131".TrigDFT;
	::Energiemes:apModulEnergie.EnabEnergy AT %QX."X20AP3131".EnabEnergy;
	::Energiemes:apModulEnergie.ClearEnergy AT %QX."X20AP3131".ClearEnergy;
	::Energiemes:apModulEnergie.ForceEnergy AT %QX."X20AP3131".ForceEnergy;
	::io307:cmModul10.di01 AT %IX."X20CM8281c".DigitalInput01;
	::io307:cmModul10.di02 AT %IX."X20CM8281c".DigitalInput02;
	::io307:cmModul10.di03 AT %IX."X20CM8281c".DigitalInput03;
	::io307:cmModul10.di04 AT %IX."X20CM8281c".DigitalInput04;
	::io307:cmModul10.do01 AT %QX."X20CM8281c".DigitalOutput01;
	::io307:cmModul10.do02 AT %QX."X20CM8281c".DigitalOutput02;
	::io307:cmModul10.ai01 AT %IW."X20CM8281c".AnalogInput01;
	::io307:cmModul10.ao01 AT %QW."X20CM8281c".AnalogOutput01;
	::io307:cmModul10.StatusInput01 AT %IB."X20CM8281c".StatusInput01;
	::io307:cmModul11.di01 AT %IX."X20CM8281d".DigitalInput01;
	::io307:cmModul11.di02 AT %IX."X20CM8281d".DigitalInput02;
	::io307:cmModul11.di03 AT %IX."X20CM8281d".DigitalInput03;
	::io307:cmModul11.di04 AT %IX."X20CM8281d".DigitalInput04;
	::io307:cmModul11.do01 AT %QX."X20CM8281d".DigitalOutput01;
	::io307:cmModul11.do02 AT %QX."X20CM8281d".DigitalOutput02;
	::io307:cmModul11.ai01 AT %IW."X20CM8281d".AnalogInput01;
	::io307:cmModul11.ao01 AT %QW."X20CM8281d".AnalogOutput01;
	::io307:cmModul11.StatusInput01 AT %IB."X20CM8281d".StatusInput01;
	::io307:brModul01.ModulOk AT %IX."X20BR7300".IF1.ST1.ModuleOk;
	::io307:diModul02.ModulOk AT %IX."X20DIF371".ModuleOk;
	::io307:doModul03.ModulOk AT %IX."X20DO9322".ModuleOk;
	::io307:aiModul04.ModulOk AT %IX."X20AI8321".ModuleOk;
	::io307:cmModul05.ModulOk AT %IX."X20CM8281".ModuleOk;
	::io307:cmModul06.ModulOk AT %IX."X20CM8281a".ModuleOk;
	::io307:cmModul07.ModulOk AT %IX."X20CM8281b".ModuleOk;
	::Energiemes:apModulEnergie.ModulOk AT %IX."X20AP3131".ModuleOk;
	::io307:cmModul10.ModulOk AT %IX."X20CM8281c".ModuleOk;
	::io307:cmModul11.ModulOk AT %IX."X20CM8281d".ModuleOk;
	::io307:cmModul12.ModulOk AT %IX."X20CM8281e".ModuleOk;
	::io307:cmModul12.di01 AT %IX."X20CM8281e".DigitalInput01;
	::io307:cmModul12.di02 AT %IX."X20CM8281e".DigitalInput02;
	::io307:cmModul12.di03 AT %IX."X20CM8281e".DigitalInput03;
	::io307:cmModul12.di04 AT %IX."X20CM8281e".DigitalInput04;
	::io307:cmModul12.do01 AT %QX."X20CM8281e".DigitalOutput01;
	::io307:cmModul12.do02 AT %QX."X20CM8281e".DigitalOutput02;
	::io307:cmModul12.ai01 AT %IW."X20CM8281e".AnalogInput01;
	::io307:cmModul12.ao01 AT %QW."X20CM8281e".AnalogOutput01;
	::io307:cmModul12.StatusInput01 AT %IB."X20CM8281e".StatusInput01;
END_VAR
```

- Physical/3_07/4PPC30_0702_21B/PvMap.vvm: same as Physical/2_07/4PPC30_0702_21B/Cpu.per
- Physical/3_07/4PPC30_0702_21B/mappServices/Config.mprecipexml: same as Physical/3_04_Plus/4PPC30_043F_21B/mappServices/Config.mprecipexml
## Configuration 4_07

CPU 4PPC30.0702-21B, AutomationRuntime S4.93, Build 4.1.2, Vc V4.73.5

### Task classes (Cpu.sw)
```
Cyclic#1 (cycle 10000 us, tolerance 10000 us):
  eUhr <- Util.eUhr.prg
  UsbLink <- CSV.UsbLink.prg
Cyclic#2 (cycle 20000 us, tolerance 20000 us):
  hmiMain <- Visualisierung.hmiMain.prg
  System <- Util.System.prg
  StartStopp <- Steuerung.StartStopp.prg
  mappPara <- Util.mappPara.prg
Cyclic#3 (cycle 50000 us, tolerance 50000 us):
  io407 <- IO.io407.prg
  aktorenMap <- IO.aktorenMapping.prg
  boxenMappi <- IO.boxenMapping.prg
  Ablaufstrg <- Ablaufsteuerung.Ablaufstrg.prg
  Leistung <- Regelung.Leistung.prg
  Sitemanage <- Sitemanager.Sitemanager.prg
Cyclic#4 (cycle 100000 us, tolerance 100000 us):
  Nutzung <- Util.Nutzung.prg
  Alarm <- Alarmsystem.Alarm.prg
  Berechnung <- Berechnung.Berechnung.prg
Cyclic#5 (cycle 200000 us, tolerance 200000 us):
  Energiemes <- IO.Energiemessung.prg
  hmiConnect <- Visualisierung.hmiConnect.prg
Cyclic#6 (cycle 500000 us, tolerance 500000 us):
  CSV01_EXT <- CSV.CSV01_EXT.prg
  CSV01_PRG <- CSV.CSV01_PRG.prg
DataObjects: CSV01_CFG <- CSV.CSV01_CFG.dob
VcDataObjects: Visu <- Visualisierung.Visu.dob
Binaries: vccddbox, vccbtn, vcpdvnc, arialbd, vcmgr, vctcal, vcgclass, vcfile, vccnum, TCData, vcfntttf, vcpkat, vcdsloc, vcbclass, udbdef, FWRules, vcpd335x, vccstr, vccalarm, visvc, arial, Visu03, vccshape, vcalarm, vcpfppct, Visu01, vccdt, vcptelo, vcchspot, vcpk, vccbmp, vccpopup, vcshared, vcrt, vcnet, Visu02, vcctext, vcctrend, arsvcreg, vcclbox, vccbar, vcdsint, vcpdsw, vccovl, vccline, Config, sysconf, Role, User, ashwd, ashwac, iomap, arconfig, asfw
Libraries: operator, runtime, astime, AsIecCon, standard, sys_lib, AsBrStr, LascoMath, LascoReg, LascoTrock, LascoUtil, LaEntfV2, LascoBoxen, LoopConR, brsystem, asstring, FileIO, DataObj, AsARCfg, visapi, AsUSB, dvframe, IecCheck, AsTCP, MpRecipe, MpBase, MpFile, CSV, vcresman, CControl
```

### Hardware
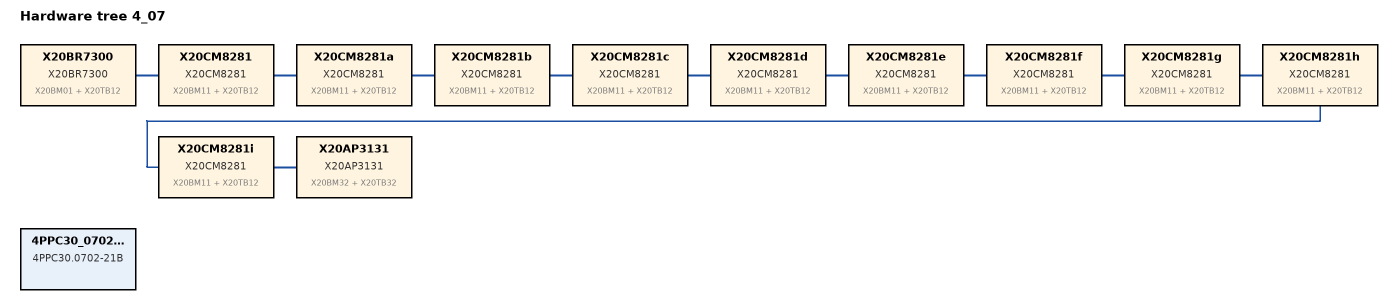
```
4PPC30_0702_21B : 4PPC30.0702-21B v1.1.4.0
  Connector IF3:
    ActivateDevice = 1
    Mode = Manual
    InternetAddress = 10.0.0.2
    SubnetMask = 255.255.255.0
    Vnc1
    VncVcObjectName1 = Visu
    VncKeyMappingFile1 = VC\PS2-Keyboard.dis
    VncMaxConnections1 = 5
    VncRefreshRate1 = 100
  Connector IF4:
    TerminatingResistor = 1
  ConfigurationID = CControl407Plus_4_07
  UserPartitionSize = 300
  RemanentGlobalPvSize = 7200
  EnableUsbRemoteInstall = 1
  TimerDeviceType = SWIOTIMER
  Cyclic1Duration = 10000
  Cyclic1Tolerance = 10000
  Cyclic2Duration = 20000
  Cyclic2Tolerance = 20000
  Cyclic3Duration = 50000
  Cyclic3Tolerance = 50000
  Cyclic4Duration = 100000
  Cyclic4Tolerance = 100000
  Cyclic5Duration = 200000
  Cyclic5Tolerance = 200000
  Cyclic6Duration = 500000
  Cyclic6Tolerance = 500000
  Cyclic7Duration = 1000000
  Cyclic7Tolerance = 1000000
  Cyclic8Duration = 10000
  Cyclic8Tolerance = 30000000
  FileDevice1
  FileDeviceName1 = CF
  FileDevicePath1 = F:\
  FileDevice2
  FileDeviceName2 = 
  FileDevicePath2 = 
  TimeZone = 140
  ActivateDaylightSavingTime = 1
  FtpUser1
  FtpUsername1 = lasco
  FtpUserPassword1 = SNwwCTsxQArJwbBFpOip1xSm5gs084piIrpMjK5ODJk=
  FtpUserSalt1 = KOYStMs7
  FTPAccessRight1 = 0
  FTPdevice1 = ALL
  VcObjectName = Visu
  KeyMappingFile = VC\4PPC30_0702_21B.dis
X20AP3131 : X20AP3131 v1.5.0.0  [SS1 -> X20TB32.SS; SL -> X20BM32.SL1]
  FunctionModel = CANIOBusController
  Supervision = off
  CurrentRatioA = 50
  CurrentRatioB = 50
  CurrentRatioC = 50
X20BM01 : X20BM01 v2.2.0.0
X20BM11 : X20BM11 v1.1.0.0  [X2X1 -> X20BM01.IF1]
X20BM11a : X20BM11 v1.1.0.0  [X2X1 -> X20BM11.X2X2]
X20BM11b : X20BM11 v1.1.0.0  [X2X1 -> X20BM11a.X2X2]
X20BM11c : X20BM11 v1.1.0.0  [X2X1 -> X20BM11b.X2X2]
X20BM11d : X20BM11 v1.1.0.0  [X2X1 -> X20BM11c.X2X2]
X20BM11e : X20BM11 v1.1.0.0  [X2X1 -> X20BM11d.X2X2]
X20BM11f : X20BM11 v1.1.0.0  [X2X1 -> X20BM11e.X2X2]
X20BM11g : X20BM11 v1.1.0.0  [X2X1 -> X20BM11f.X2X2]
X20BM11h : X20BM11 v1.1.0.0  [X2X1 -> X20BM11g.X2X2]
X20BM11i : X20BM11 v1.1.0.0  [X2X1 -> X20BM11h.X2X2]
X20BM32 : X20BM32 v1.1.0.0  [X2X1 -> X20BM11i.X2X2]
X20BR7300 : X20BR7300 v1.7.0.0  [CAN1 -> 4PPC30_0702_21B.IF4; SL -> X20BM01.SL1; SS1 -> X20TB12.SS]
  Supervision = off
X20CM8281 : X20CM8281 v1.4.0.0  [SS1 -> X20TB12a.SS; SL -> X20BM11.SL1]
  FunctionModel = CANIOBusController
  Supervision = off
  ChannelType01AI = 4 to 20mA
  LowerLimitAI = 0
  ChannelType01AO = 0 to 20mA
X20CM8281a : X20CM8281 v1.4.0.0  [SS1 -> X20TB12b.SS; SL -> X20BM11a.SL1]
  FunctionModel = CANIOBusController
  Supervision = off
  ChannelType01AI = 4 to 20mA
  LowerLimitAI = 0
  ChannelType01AO = 0 to 20mA
X20CM8281b : X20CM8281 v1.4.0.0  [SS1 -> X20TB12c.SS; SL -> X20BM11b.SL1]
  FunctionModel = CANIOBusController
  Supervision = off
  ChannelType01AI = 4 to 20mA
  LowerLimitAI = 0
  ChannelType01AO = 0 to 20mA
X20CM8281c : X20CM8281 v1.4.0.0  [SS1 -> X20TB12d.SS; SL -> X20BM11c.SL1]
  FunctionModel = CANIOBusController
  Supervision = off
  ChannelType01AI = 4 to 20mA
  LowerLimitAI = 0
X20CM8281d : X20CM8281 v1.4.0.0  [SS1 -> X20TB12e.SS; SL -> X20BM11d.SL1]
  FunctionModel = CANIOBusController
  Supervision = off
  ChannelType01AI = 4 to 20mA
  LowerLimitAI = 0
X20CM8281e : X20CM8281 v1.4.0.0  [SS1 -> X20TB12f.SS; SL -> X20BM11e.SL1]
  FunctionModel = CANIOBusController
  Supervision = off
  ChannelType01AI = 4 to 20mA
  LowerLimitAI = 0
X20CM8281f : X20CM8281 v1.4.0.0  [SS1 -> X20TB12g.SS; SL -> X20BM11f.SL1]
  FunctionModel = CANIOBusController
  Supervision = off
  ChannelType01AI = 4 to 20mA
  LowerLimitAI = 0
  ChannelType01AO = 0 to 20mA
X20CM8281g : X20CM8281 v1.4.0.0  [SS1 -> X20TB12h.SS; SL -> X20BM11g.SL1]
  FunctionModel = CANIOBusController
  Supervision = off
  ChannelType01AI = 4 to 20mA
  LowerLimitAI = 0
X20CM8281h : X20CM8281 v1.4.0.0  [SS1 -> X20TB12i.SS; SL -> X20BM11h.SL1]
  FunctionModel = CANIOBusController
  Supervision = off
X20CM8281i : X20CM8281 v1.4.0.0  [SS1 -> X20TB12j.SS; SL -> X20BM11i.SL1]
  FunctionModel = CANIOBusController
  Supervision = off
  ChannelType01AI = 4 to 20mA
X20TB12 : X20TB12 v1.0.0.0
X20TB12a : X20TB12 v1.0.0.0
X20TB12b : X20TB12 v1.0.0.0
X20TB12c : X20TB12 v1.0.0.0
X20TB12d : X20TB12 v1.0.0.0
X20TB12e : X20TB12 v1.0.0.0
X20TB12f : X20TB12 v1.0.0.0
X20TB12g : X20TB12 v1.0.0.0
X20TB12h : X20TB12 v1.0.0.0
X20TB12i : X20TB12 v1.0.0.0
X20TB12j : X20TB12 v1.0.0.0
X20TB32 : X20TB32 v1.0.0.1
```

- Physical/4_07/4PPC30_0702_21B/Cpu.per: same as Physical/2_07/4PPC30_0702_21B/Cpu.per
### IoMap.iom - 4PPC30_0702_21B/IoMap.iom
```iecst
VAR_CONFIG
	::io407:cmModul02.di01 AT %IX."X20CM8281".DigitalInput01;
	::io407:cmModul02.di02 AT %IX."X20CM8281".DigitalInput02;
	::io407:cmModul02.di03 AT %IX."X20CM8281".DigitalInput03;
	::io407:cmModul02.di04 AT %IX."X20CM8281".DigitalInput04;
	::io407:cmModul02.do01 AT %QX."X20CM8281".DigitalOutput01;
	::io407:cmModul02.do02 AT %QX."X20CM8281".DigitalOutput02;
	::io407:cmModul02.ai01 AT %IW."X20CM8281".AnalogInput01;
	::io407:cmModul02.ao01 AT %QW."X20CM8281".AnalogOutput01;
	::io407:cmModul02.StatusInput01 AT %IB."X20CM8281".StatusInput01;
	::io407:cmModul03.di01 AT %IX."X20CM8281a".DigitalInput01;
	::io407:cmModul03.di02 AT %IX."X20CM8281a".DigitalInput02;
	::io407:cmModul03.di03 AT %IX."X20CM8281a".DigitalInput03;
	::io407:cmModul03.di04 AT %IX."X20CM8281a".DigitalInput04;
	::io407:cmModul03.do01 AT %QX."X20CM8281a".DigitalOutput01;
	::io407:cmModul03.do02 AT %QX."X20CM8281a".DigitalOutput02;
	::io407:cmModul03.ai01 AT %IW."X20CM8281a".AnalogInput01;
	::io407:cmModul03.ao01 AT %QW."X20CM8281a".AnalogOutput01;
	::io407:cmModul03.StatusInput01 AT %IB."X20CM8281a".StatusInput01;
	::io407:cmModul04.di01 AT %IX."X20CM8281b".DigitalInput01;
	::io407:cmModul04.di02 AT %IX."X20CM8281b".DigitalInput02;
	::io407:cmModul04.di03 AT %IX."X20CM8281b".DigitalInput03;
	::io407:cmModul04.di04 AT %IX."X20CM8281b".DigitalInput04;
	::io407:cmModul04.do01 AT %QX."X20CM8281b".DigitalOutput01;
	::io407:cmModul04.do02 AT %QX."X20CM8281b".DigitalOutput02;
	::io407:cmModul04.ai01 AT %IW."X20CM8281b".AnalogInput01;
	::io407:cmModul04.ao01 AT %QW."X20CM8281b".AnalogOutput01;
	::io407:cmModul04.StatusInput01 AT %IB."X20CM8281b".StatusInput01;
	::io407:cmModul05.di01 AT %IX."X20CM8281c".DigitalInput01;
	::io407:cmModul05.di02 AT %IX."X20CM8281c".DigitalInput02;
	::io407:cmModul05.di03 AT %IX."X20CM8281c".DigitalInput03;
	::io407:cmModul05.di04 AT %IX."X20CM8281c".DigitalInput04;
	::io407:cmModul05.do01 AT %QX."X20CM8281c".DigitalOutput01;
	::io407:cmModul05.do02 AT %QX."X20CM8281c".DigitalOutput02;
	::io407:cmModul05.ai01 AT %IW."X20CM8281c".AnalogInput01;
	::io407:cmModul05.ao01 AT %QW."X20CM8281c".AnalogOutput01;
	::io407:cmModul05.StatusInput01 AT %IB."X20CM8281c".StatusInput01;
	::io407:cmModul06.di01 AT %IX."X20CM8281d".DigitalInput01;
	::io407:cmModul06.di02 AT %IX."X20CM8281d".DigitalInput02;
	::io407:cmModul06.di03 AT %IX."X20CM8281d".DigitalInput03;
	::io407:cmModul06.di04 AT %IX."X20CM8281d".DigitalInput04;
	::io407:cmModul06.do01 AT %QX."X20CM8281d".DigitalOutput01;
	::io407:cmModul06.do02 AT %QX."X20CM8281d".DigitalOutput02;
	::io407:cmModul06.ai01 AT %IW."X20CM8281d".AnalogInput01;
	::io407:cmModul06.ao01 AT %QW."X20CM8281d".AnalogOutput01;
	::io407:cmModul06.StatusInput01 AT %IB."X20CM8281d".StatusInput01;
	::io407:cmModul07.di01 AT %IX."X20CM8281e".DigitalInput01;
	::io407:cmModul07.di02 AT %IX."X20CM8281e".DigitalInput02;
	::io407:cmModul07.di03 AT %IX."X20CM8281e".DigitalInput03;
	::io407:cmModul07.di04 AT %IX."X20CM8281e".DigitalInput04;
	::io407:cmModul07.do01 AT %QX."X20CM8281e".DigitalOutput01;
	::io407:cmModul07.do02 AT %QX."X20CM8281e".DigitalOutput02;
	::io407:cmModul07.ai01 AT %IW."X20CM8281e".AnalogInput01;
	::io407:cmModul07.ao01 AT %QW."X20CM8281e".AnalogOutput01;
	::io407:cmModul07.StatusInput01 AT %IB."X20CM8281e".StatusInput01;
	::io407:cmModul08.di01 AT %IX."X20CM8281f".DigitalInput01;
	::io407:cmModul08.di02 AT %IX."X20CM8281f".DigitalInput02;
	::io407:cmModul08.di03 AT %IX."X20CM8281f".DigitalInput03;
	::io407:cmModul08.di04 AT %IX."X20CM8281f".DigitalInput04;
	::io407:cmModul08.do01 AT %QX."X20CM8281f".DigitalOutput01;
	::io407:cmModul08.do02 AT %QX."X20CM8281f".DigitalOutput02;
	::io407:cmModul08.ai01 AT %IW."X20CM8281f".AnalogInput01;
	::io407:cmModul08.ao01 AT %QW."X20CM8281f".AnalogOutput01;
	::io407:cmModul08.StatusInput01 AT %IB."X20CM8281f".StatusInput01;
	::io407:cmModul09.di01 AT %IX."X20CM8281g".DigitalInput01;
	::io407:cmModul09.di02 AT %IX."X20CM8281g".DigitalInput02;
	::io407:cmModul09.di03 AT %IX."X20CM8281g".DigitalInput03;
	::io407:cmModul09.di04 AT %IX."X20CM8281g".DigitalInput04;
	::io407:cmModul09.do01 AT %QX."X20CM8281g".DigitalOutput01;
	::io407:cmModul09.do02 AT %QX."X20CM8281g".DigitalOutput02;
	::io407:cmModul09.ai01 AT %IW."X20CM8281g".AnalogInput01;
	::io407:cmModul09.ao01 AT %QW."X20CM8281g".AnalogOutput01;
	::io407:cmModul09.StatusInput01 AT %IB."X20CM8281g".StatusInput01;
	::io407:cmModul10.di01 AT %IX."X20CM8281h".DigitalInput01;
	::io407:cmModul10.di02 AT %IX."X20CM8281h".DigitalInput02;
	::io407:cmModul10.di03 AT %IX."X20CM8281h".DigitalInput03;
	::io407:cmModul10.di04 AT %IX."X20CM8281h".DigitalInput04;
	::io407:cmModul10.do01 AT %QX."X20CM8281h".DigitalOutput01;
	::io407:cmModul10.do02 AT %QX."X20CM8281h".DigitalOutput02;
	::io407:cmModul10.ai01 AT %IW."X20CM8281h".AnalogInput01;
	::io407:cmModul10.ao01 AT %QW."X20CM8281h".AnalogOutput01;
	::io407:cmModul10.StatusInput01 AT %IB."X20CM8281h".StatusInput01;
	::io407:cmModul11.di01 AT %IX."X20CM8281i".DigitalInput01;
	::io407:cmModul11.di02 AT %IX."X20CM8281i".DigitalInput02;
	::io407:cmModul11.di03 AT %IX."X20CM8281i".DigitalInput03;
	::io407:cmModul11.di04 AT %IX."X20CM8281i".DigitalInput04;
	::io407:cmModul11.do01 AT %QX."X20CM8281i".DigitalOutput01;
	::io407:cmModul11.do02 AT %QX."X20CM8281i".DigitalOutput02;
	::io407:cmModul11.ai01 AT %IW."X20CM8281i".AnalogInput01;
	::io407:cmModul11.ao01 AT %QW."X20CM8281i".AnalogOutput01;
	::io407:cmModul11.StatusInput01 AT %IB."X20CM8281i".StatusInput01;
	::Energiemes:apModulEnergie.PmeanT AT %IW."X20AP3131".PmeanT;
	::Energiemes:apModulEnergie.QmeanT AT %IW."X20AP3131".QmeanT;
	::Energiemes:apModulEnergie.SmeanT AT %IW."X20AP3131".SmeanT;
	::Energiemes:apModulEnergie.PFmeanT AT %IW."X20AP3131".PFmeanT;
	::Energiemes:apModulEnergie.AenergyT AT %ID."X20AP3131".AenergyT;
	::Energiemes:apModulEnergie.RenergyT AT %ID."X20AP3131".RenergyT;
	::Energiemes:apModulEnergie.SAenergyT AT %ID."X20AP3131".SAenergyT;
	::Energiemes:apModulEnergie.RBClearEnergy AT %IX."X20AP3131".RBClearEnergy;
	::Energiemes:apModulEnergie.TrigDFT AT %QX."X20AP3131".TrigDFT;
	::Energiemes:apModulEnergie.EnabEnergy AT %QX."X20AP3131".EnabEnergy;
	::Energiemes:apModulEnergie.ClearEnergy AT %QX."X20AP3131".ClearEnergy;
	::Energiemes:apModulEnergie.ForceEnergy AT %QX."X20AP3131".ForceEnergy;
	::io407:brModul01.ModulOk AT %IX."X20BR7300".IF1.ST1.ModuleOk;
	::io407:cmModul02.ModulOk AT %IX."X20CM8281".ModuleOk;
	::io407:cmModul03.ModulOk AT %IX."X20CM8281a".ModuleOk;
	::io407:cmModul04.ModulOk AT %IX."X20CM8281b".ModuleOk;
	::io407:cmModul05.ModulOk AT %IX."X20CM8281c".ModuleOk;
	::io407:cmModul06.ModulOk AT %IX."X20CM8281d".ModuleOk;
	::io407:cmModul07.ModulOk AT %IX."X20CM8281e".ModuleOk;
	::io407:cmModul08.ModulOk AT %IX."X20CM8281f".ModuleOk;
	::io407:cmModul09.ModulOk AT %IX."X20CM8281g".ModuleOk;
	::io407:cmModul10.ModulOk AT %IX."X20CM8281h".ModuleOk;
	::io407:cmModul11.ModulOk AT %IX."X20CM8281i".ModuleOk;
	::Energiemes:apModulEnergie.ModulOk AT %IX."X20AP3131".ModuleOk;
END_VAR
```

- Physical/4_07/4PPC30_0702_21B/mappServices/Config.mprecipexml: same as Physical/2_07/4PPC30_0702_21B/mappServices/Config.mprecipexml
## Configuration 4_07_Plus

CPU 4PPC30.0702-21B, AutomationRuntime S4.93, Build 4.1.2, Safety 0.0, Vc V4.73.5

### Task classes (Cpu.sw)
```
Cyclic#1 (cycle 10000 us, tolerance 10000 us):
  eUhr <- Util.eUhr.prg
  UsbLink <- CSV.UsbLink.prg
Cyclic#2 (cycle 20000 us, tolerance 20000 us):
  hmiMain <- Visualisierung.hmiMain.prg
  System <- Util.System.prg
  StartStopp <- Steuerung.StartStopp.prg
  mappPara <- Util.mappPara.prg
Cyclic#3 (cycle 50000 us, tolerance 50000 us):
  io407Plus <- IO.io407Plus.prg
  aktorenMap <- IO.aktorenMapping.prg
  boxenMappi <- IO.boxenMapping.prg
  Ablaufstrg <- Ablaufsteuerung.Ablaufstrg.prg
  Leistung <- Regelung.Leistung.prg
  Sitemanage <- Sitemanager.Sitemanager.prg
Cyclic#4 (cycle 100000 us, tolerance 100000 us):
  Nutzung <- Util.Nutzung.prg
  Alarm <- Alarmsystem.Alarm.prg
  Berechnung <- Berechnung.Berechnung.prg
Cyclic#5 (cycle 200000 us, tolerance 200000 us):
  Energiemes <- IO.Energiemessung.prg
  hmiConnect <- Visualisierung.hmiConnect.prg
Cyclic#6 (cycle 500000 us, tolerance 500000 us):
  CSV01_EXT <- CSV.CSV01_EXT.prg
  CSV01_PRG <- CSV.CSV01_PRG.prg
DataObjects: CSV01_CFG <- CSV.CSV01_CFG.dob
VcDataObjects: Visu <- Visualisierung.Visu.dob
Binaries: vccddbox, vccbtn, vcpdvnc, arialbd, vcmgr, vctcal, vcgclass, vcfile, vccnum, TCData, vcfntttf, vcpkat, vcdsloc, vcbclass, udbdef, FWRules, vcpd335x, vccstr, vccalarm, visvc, arial, Visu03, vccshape, vcalarm, vcpfppct, Visu01, vccdt, vcptelo, vcchspot, vcpk, vccbmp, vccpopup, vcshared, vcrt, vcnet, Visu02, vcctext, vcctrend, arsvcreg, vcclbox, vccbar, vcdsint, vcpdsw, vccovl, vccline, Config, sysconf, Role, User, ashwd, ashwac, iomap, arconfig, asfw
Libraries: operator, runtime, astime, AsIecCon, standard, sys_lib, AsBrStr, LascoMath, LascoReg, LascoTrock, LascoUtil, LaEntfV2, LascoBoxen, LoopConR, brsystem, asstring, FileIO, DataObj, AsARCfg, visapi, AsUSB, dvframe, IecCheck, AsTCP, MpRecipe, MpBase, MpFile, CSV, vcresman, CControl
```

### Hardware
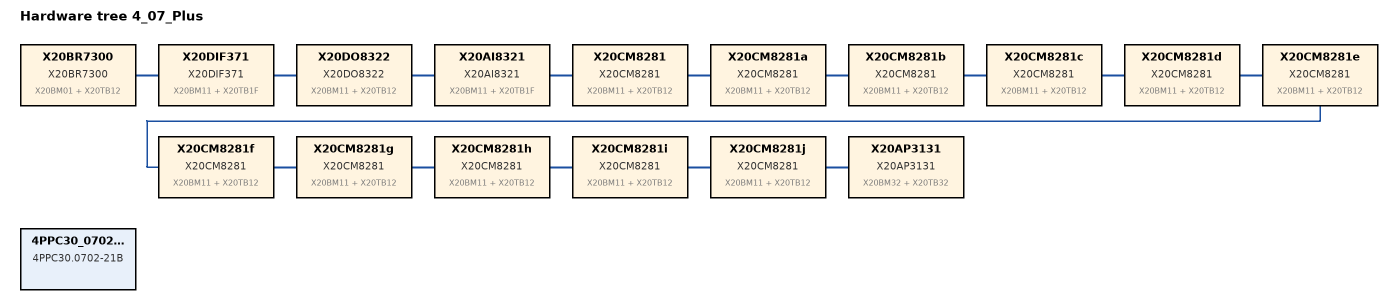
```
4PPC30_0702_21B : 4PPC30.0702-21B v1.1.4.0
  Connector IF3:
    ActivateDevice = 1
    Mode = Manual
    InternetAddress = 10.0.0.2
    SubnetMask = 255.255.255.0
    Vnc1
    VncVcObjectName1 = Visu
    VncKeyMappingFile1 = VC\PS2-Keyboard.dis
    VncMaxConnections1 = 5
    VncRefreshRate1 = 100
  Connector IF4:
    TerminatingResistor = 1
  ConfigurationID = CControl407Plus_4_07_Plus
  UserPartitionSize = 300
  RemanentGlobalPvSize = 6000
  EnableUsbRemoteInstall = 1
  TimerDeviceType = SWIOTIMER
  Cyclic1Duration = 10000
  Cyclic1Tolerance = 10000
  Cyclic2Duration = 20000
  Cyclic2Tolerance = 20000
  Cyclic3Duration = 50000
  Cyclic3Tolerance = 50000
  Cyclic4Duration = 100000
  Cyclic4Tolerance = 100000
  Cyclic5Duration = 200000
  Cyclic5Tolerance = 200000
  Cyclic6Duration = 500000
  Cyclic6Tolerance = 500000
  Cyclic7Duration = 1000000
  Cyclic7Tolerance = 1000000
  Cyclic8Duration = 10000
  Cyclic8Tolerance = 30000000
  FileDevice1
  FileDeviceName1 = CF
  FileDevicePath1 = F:\
  TimeZone = 140
  ActivateDaylightSavingTime = 1
  FtpUser1
  FtpUsername1 = lasco
  FtpUserPassword1 = eB4qta04aQSN3hSQ/CYLDrPGprp3b5FE/XWpIbl7CMk=
  FtpUserSalt1 = 2eeAO8dH
  FTPAccessRight1 = 0
  FTPdevice1 = ALL
  VcObjectName = Visu
  KeyMappingFile = VC\4PPC30_0702_21B.dis
X20AI8321 : X20AI8321 v1.5.0.0  [SS1 -> X20TB1F1.SS; SL -> X20BM11b.SL1]
  FunctionModel = CANIOBusController
  Supervision = off
  LowerLimit = 0
  ChannelType01 = 4 to 20mA
  ChannelType02 = 4 to 20mA
  ChannelType03 = 4 to 20mA
  ChannelType04 = 4 to 20mA
  ChannelType05 = 4 to 20mA
  ChannelType06 = 4 to 20mA
  ChannelType07 = 4 to 20mA
  ChannelType08 = 4 to 20mA
X20AP3131 : X20AP3131 v1.5.0.0  [SS1 -> X20TB32.SS; SL -> X20BM32.SL1]
  FunctionModel = CANIOBusController
  Supervision = off
  CurrentRatioA = 50
  CurrentRatioB = 50
  CurrentRatioC = 50
X20BM01 : X20BM01 v2.2.0.0
X20BM11 : X20BM11 v1.1.0.0  [X2X1 -> X20BM01.IF1]
X20BM11a : X20BM11 v1.1.0.0  [X2X1 -> X20BM11.X2X2]
X20BM11b : X20BM11 v1.1.0.0  [X2X1 -> X20BM11a.X2X2]
X20BM11c : X20BM11 v1.1.0.0  [X2X1 -> X20BM11b.X2X2]
X20BM11d : X20BM11 v1.1.0.0  [X2X1 -> X20BM11c.X2X2]
X20BM11e : X20BM11 v1.1.0.0  [X2X1 -> X20BM11d.X2X2]
X20BM11f : X20BM11 v1.1.0.0  [X2X1 -> X20BM11e.X2X2]
X20BM11g : X20BM11 v1.1.0.0  [X2X1 -> X20BM11f.X2X2]
X20BM11h : X20BM11 v1.1.0.0  [X2X1 -> X20BM11g.X2X2]
X20BM11i : X20BM11 v1.1.0.0  [X2X1 -> X20BM11h.X2X2]
X20BM11j : X20BM11 v1.1.0.0  [X2X1 -> X20BM11i.X2X2]
X20BM11k : X20BM11 v1.1.0.0  [X2X1 -> X20BM11j.X2X2]
X20BM11l : X20BM11 v1.1.0.0  [X2X1 -> X20BM11k.X2X2]
X20BM11m : X20BM11 v1.1.0.0  [X2X1 -> X20BM11l.X2X2]
X20BM32 : X20BM32 v1.1.0.0  [X2X1 -> X20BM11m.X2X2]
X20BR7300 : X20BR7300 v1.7.0.0  [CAN1 -> 4PPC30_0702_21B.IF4; SL -> X20BM01.SL1; SS1 -> X20TB12.SS]
  Supervision = off
X20CM8281 : X20CM8281 v1.4.0.0  [SS1 -> X20TB12b.SS; SL -> X20BM11c.SL1]
  FunctionModel = CANIOBusController
  Supervision = off
  ChannelType01AO = 0 to 20mA
X20CM8281a : X20CM8281 v1.4.0.0  [SS1 -> X20TB12c.SS; SL -> X20BM11d.SL1]
  FunctionModel = CANIOBusController
  Supervision = off
  ChannelType01AI = 4 to 20mA
  LowerLimitAI = 0
  ChannelType01AO = 0 to 20mA
X20CM8281b : X20CM8281 v1.4.0.0  [SS1 -> X20TB12d.SS; SL -> X20BM11e.SL1]
  FunctionModel = CANIOBusController
  Supervision = off
  ChannelType01AI = 4 to 20mA
  LowerLimitAI = 0
  ChannelType01AO = 0 to 20mA
X20CM8281c : X20CM8281 v1.4.0.0  [SS1 -> X20TB12e.SS; SL -> X20BM11f.SL1]
  FunctionModel = CANIOBusController
  Supervision = off
  ChannelType01AI = 4 to 20mA
  LowerLimitAI = 0
  ChannelType01AO = 0 to 20mA
X20CM8281d : X20CM8281 v1.4.0.0  [SS1 -> X20TB12f.SS; SL -> X20BM11g.SL1]
  FunctionModel = CANIOBusController
  Supervision = off
  ChannelType01AI = 4 to 20mA
  LowerLimitAI = 0
  ChannelType01AO = 0 to 20mA
X20CM8281e : X20CM8281 v1.4.0.0  [SS1 -> X20TB12g.SS; SL -> X20BM11h.SL1]
  FunctionModel = CANIOBusController
  Supervision = off
  ChannelType01AI = 4 to 20mA
  LowerLimitAI = 0
X20CM8281f : X20CM8281 v1.4.0.0  [SS1 -> X20TB12h.SS; SL -> X20BM11i.SL1]
  FunctionModel = CANIOBusController
  Supervision = off
  ChannelType01AI = 4 to 20mA
  LowerLimitAI = 0
  ChannelType01AO = 0 to 20mA
X20CM8281g : X20CM8281 v1.4.0.0  [SS1 -> X20TB12i.SS; SL -> X20BM11j.SL1]
  FunctionModel = CANIOBusController
  Supervision = off
  ChannelType01AI = 4 to 20mA
  LowerLimitAI = 0
  ChannelType01AO = 0 to 20mA
X20CM8281h : X20CM8281 v1.4.0.0  [SS1 -> X20TB12j.SS; SL -> X20BM11k.SL1]
  FunctionModel = CANIOBusController
  Supervision = off
  ChannelType01AI = 4 to 20mA
  LowerLimitAI = 0
  ChannelType01AO = 0 to 20mA
X20CM8281i : X20CM8281 v1.4.0.0  [SS1 -> X20TB12k.SS; SL -> X20BM11l.SL1]
  FunctionModel = CANIOBusController
  Supervision = off
  ChannelType01AI = 4 to 20mA
  LowerLimitAI = 0
  ChannelType01AO = 0 to 20mA
X20CM8281j : X20CM8281 v1.4.0.0  [SS1 -> X20TB12l.SS; SL -> X20BM11m.SL1]
  FunctionModel = CANIOBusController
  Supervision = off
  ChannelType01AI = 4 to 20mA
  ChannelType01AO = 0 to 20mA
X20DIF371 : X20DIF371 v1.3.0.0  [SS1 -> X20TB1F.SS; SL -> X20BM11.SL1]
  FunctionModel = CANIOBusController
  Supervision = off
X20DO8322 : X20DO8322 v1.5.0.0  [SS1 -> X20TB12a.SS; SL -> X20BM11a.SL1]
  FunctionModel = CANIOBusController
  Supervision = off
X20TB12 : X20TB12 v1.0.0.0
X20TB12a : X20TB12 v1.0.0.0
X20TB12b : X20TB12 v1.0.0.0
X20TB12c : X20TB12 v1.0.0.0
X20TB12d : X20TB12 v1.0.0.0
X20TB12e : X20TB12 v1.0.0.0
X20TB12f : X20TB12 v1.0.0.0
X20TB12g : X20TB12 v1.0.0.0
X20TB12h : X20TB12 v1.0.0.0
X20TB12i : X20TB12 v1.0.0.0
X20TB12j : X20TB12 v1.0.0.0
X20TB12k : X20TB12 v1.0.0.0
X20TB12l : X20TB12 v1.0.0.0
X20TB1F : X20TB1F v1.0.0.0
X20TB1F1 : X20TB1F v1.0.0.0
X20TB32 : X20TB32 v1.0.0.1
```

- Physical/4_07_Plus/4PPC30_0702_21B/Cpu.per: same as Physical/2_07/4PPC30_0702_21B/Cpu.per
### IoMap.iom - 4PPC30_0702_21B/IoMap.iom
```iecst
VAR_CONFIG
	::io407Plus:diModul02.di01 AT %IX."X20DIF371".DigitalInput01;
	::io407Plus:diModul02.di02 AT %IX."X20DIF371".DigitalInput02;
	::io407Plus:diModul02.di03 AT %IX."X20DIF371".DigitalInput03;
	::io407Plus:diModul02.di04 AT %IX."X20DIF371".DigitalInput04;
	::io407Plus:diModul02.di05 AT %IX."X20DIF371".DigitalInput05;
	::io407Plus:diModul02.di06 AT %IX."X20DIF371".DigitalInput06;
	::io407Plus:diModul02.di07 AT %IX."X20DIF371".DigitalInput07;
	::io407Plus:diModul02.di08 AT %IX."X20DIF371".DigitalInput08;
	::io407Plus:diModul02.di09 AT %IX."X20DIF371".DigitalInput09;
	::io407Plus:diModul02.di10 AT %IX."X20DIF371".DigitalInput10;
	::io407Plus:diModul02.di11 AT %IX."X20DIF371".DigitalInput11;
	::io407Plus:diModul02.di12 AT %IX."X20DIF371".DigitalInput12;
	::io407Plus:diModul02.di13 AT %IX."X20DIF371".DigitalInput13;
	::io407Plus:diModul02.di14 AT %IX."X20DIF371".DigitalInput14;
	::io407Plus:diModul02.di15 AT %IX."X20DIF371".DigitalInput15;
	::io407Plus:diModul02.di16 AT %IX."X20DIF371".DigitalInput16;
	::io407Plus:doModul03.do01 AT %QX."X20DO8322".DigitalOutput01;
	::io407Plus:doModul03.do02 AT %QX."X20DO8322".DigitalOutput02;
	::io407Plus:doModul03.do03 AT %QX."X20DO8322".DigitalOutput03;
	::io407Plus:doModul03.do04 AT %QX."X20DO8322".DigitalOutput04;
	::io407Plus:doModul03.do05 AT %QX."X20DO8322".DigitalOutput05;
	::io407Plus:doModul03.do06 AT %QX."X20DO8322".DigitalOutput06;
	::io407Plus:doModul03.do07 AT %QX."X20DO8322".DigitalOutput07;
	::io407Plus:doModul03.do08 AT %QX."X20DO8322".DigitalOutput08;
	::io407Plus:aiModul04.ai01 AT %IW."X20AI8321".AnalogInput01;
	::io407Plus:aiModul04.ai02 AT %IW."X20AI8321".AnalogInput02;
	::io407Plus:aiModul04.ai03 AT %IW."X20AI8321".AnalogInput03;
	::io407Plus:aiModul04.ai04 AT %IW."X20AI8321".AnalogInput04;
	::io407Plus:aiModul04.ai05 AT %IW."X20AI8321".AnalogInput05;
	::io407Plus:aiModul04.ai06 AT %IW."X20AI8321".AnalogInput06;
	::io407Plus:aiModul04.ai07 AT %IW."X20AI8321".AnalogInput07;
	::io407Plus:aiModul04.ai08 AT %IW."X20AI8321".AnalogInput08;
	::io407Plus:aiModul04.StatusInput01 AT %IB."X20AI8321".StatusInput01;
	::io407Plus:aiModul04.StatusInput02 AT %IB."X20AI8321".StatusInput02;
	::io407Plus:cmModul05.di01 AT %IX."X20CM8281".DigitalInput01;
	::io407Plus:cmModul05.di02 AT %IX."X20CM8281".DigitalInput02;
	::io407Plus:cmModul05.di03 AT %IX."X20CM8281".DigitalInput03;
	::io407Plus:cmModul05.di04 AT %IX."X20CM8281".DigitalInput04;
	::io407Plus:cmModul05.do01 AT %QX."X20CM8281".DigitalOutput01;
	::io407Plus:cmModul05.do02 AT %QX."X20CM8281".DigitalOutput02;
	::io407Plus:cmModul05.ai01 AT %IW."X20CM8281".AnalogInput01;
	::io407Plus:cmModul05.ao01 AT %QW."X20CM8281".AnalogOutput01;
	::io407Plus:cmModul05.StatusInput01 AT %IB."X20CM8281".StatusInput01;
	::io407Plus:cmModul06.di01 AT %IX."X20CM8281a".DigitalInput01;
	::io407Plus:cmModul06.di02 AT %IX."X20CM8281a".DigitalInput02;
	::io407Plus:cmModul06.di03 AT %IX."X20CM8281a".DigitalInput03;
	::io407Plus:cmModul06.di04 AT %IX."X20CM8281a".DigitalInput04;
	::io407Plus:cmModul06.do01 AT %QX."X20CM8281a".DigitalOutput01;
	::io407Plus:cmModul06.do02 AT %QX."X20CM8281a".DigitalOutput02;
	::io407Plus:cmModul06.ai01 AT %IW."X20CM8281a".AnalogInput01;
	::io407Plus:cmModul06.ao01 AT %QW."X20CM8281a".AnalogOutput01;
	::io407Plus:cmModul06.StatusInput01 AT %IB."X20CM8281a".StatusInput01;
	::io407Plus:cmModul07.di01 AT %IX."X20CM8281b".DigitalInput01;
	::io407Plus:cmModul07.di02 AT %IX."X20CM8281b".DigitalInput02;
	::io407Plus:cmModul07.di03 AT %IX."X20CM8281b".DigitalInput03;
	::io407Plus:cmModul07.di04 AT %IX."X20CM8281b".DigitalInput04;
	::io407Plus:cmModul07.do01 AT %QX."X20CM8281b".DigitalOutput01;
	::io407Plus:cmModul07.do02 AT %QX."X20CM8281b".DigitalOutput02;
	::io407Plus:cmModul07.ai01 AT %IW."X20CM8281b".AnalogInput01;
	::io407Plus:cmModul07.ao01 AT %QW."X20CM8281b".AnalogOutput01;
	::io407Plus:cmModul07.StatusInput01 AT %IB."X20CM8281b".StatusInput01;
	::io407Plus:cmModul08.di01 AT %IX."X20CM8281c".DigitalInput01;
	::io407Plus:cmModul08.di02 AT %IX."X20CM8281c".DigitalInput02;
	::io407Plus:cmModul08.di03 AT %IX."X20CM8281c".DigitalInput03;
	::io407Plus:cmModul08.di04 AT %IX."X20CM8281c".DigitalInput04;
	::io407Plus:cmModul08.do01 AT %QX."X20CM8281c".DigitalOutput01;
	::io407Plus:cmModul08.do02 AT %QX."X20CM8281c".DigitalOutput02;
	::io407Plus:cmModul08.ai01 AT %IW."X20CM8281c".AnalogInput01;
	::io407Plus:cmModul08.ao01 AT %QW."X20CM8281c".AnalogOutput01;
	::io407Plus:cmModul08.StatusInput01 AT %IB."X20CM8281c".StatusInput01;
	::io407Plus:cmModul09.di01 AT %IX."X20CM8281d".DigitalInput01;
	::io407Plus:cmModul09.di02 AT %IX."X20CM8281d".DigitalInput02;
	::io407Plus:cmModul09.di03 AT %IX."X20CM8281d".DigitalInput03;
	::io407Plus:cmModul09.di04 AT %IX."X20CM8281d".DigitalInput04;
	::io407Plus:cmModul09.do01 AT %QX."X20CM8281d".DigitalOutput01;
	::io407Plus:cmModul09.do02 AT %QX."X20CM8281d".DigitalOutput02;
	::io407Plus:cmModul09.ai01 AT %IW."X20CM8281d".AnalogInput01;
	::io407Plus:cmModul09.ao01 AT %QW."X20CM8281d".AnalogOutput01;
	::io407Plus:cmModul09.StatusInput01 AT %IB."X20CM8281d".StatusInput01;
	::io407Plus:cmModul10.di01 AT %IX."X20CM8281e".DigitalInput01;
	::io407Plus:cmModul10.di02 AT %IX."X20CM8281e".DigitalInput02;
	::io407Plus:cmModul10.di03 AT %IX."X20CM8281e".DigitalInput03;
	::io407Plus:cmModul10.di04 AT %IX."X20CM8281e".DigitalInput04;
	::io407Plus:cmModul10.do01 AT %QX."X20CM8281e".DigitalOutput01;
	::io407Plus:cmModul10.do02 AT %QX."X20CM8281e".DigitalOutput02;
	::io407Plus:cmModul10.ai01 AT %IW."X20CM8281e".AnalogInput01;
	::io407Plus:cmModul10.ao01 AT %QW."X20CM8281e".AnalogOutput01;
	::io407Plus:cmModul10.StatusInput01 AT %IB."X20CM8281e".StatusInput01;
	::io407Plus:cmModul11.di01 AT %IX."X20CM8281f".DigitalInput01;
	::io407Plus:cmModul11.di02 AT %IX."X20CM8281f".DigitalInput02;
	::io407Plus:cmModul11.di03 AT %IX."X20CM8281f".DigitalInput03;
	::io407Plus:cmModul11.di04 AT %IX."X20CM8281f".DigitalInput04;
	::io407Plus:cmModul11.do01 AT %QX."X20CM8281f".DigitalOutput01;
	::io407Plus:cmModul11.do02 AT %QX."X20CM8281f".DigitalOutput02;
	::io407Plus:cmModul11.ai01 AT %IW."X20CM8281f".AnalogInput01;
	::io407Plus:cmModul11.ao01 AT %QW."X20CM8281f".AnalogOutput01;
	::io407Plus:cmModul11.StatusInput01 AT %IB."X20CM8281f".StatusInput01;
	::io407Plus:cmModul12.di01 AT %IX."X20CM8281g".DigitalInput01;
	::io407Plus:cmModul12.di02 AT %IX."X20CM8281g".DigitalInput02;
	::io407Plus:cmModul12.di03 AT %IX."X20CM8281g".DigitalInput03;
	::io407Plus:cmModul12.di04 AT %IX."X20CM8281g".DigitalInput04;
	::io407Plus:cmModul12.do01 AT %QX."X20CM8281g".DigitalOutput01;
	::io407Plus:cmModul12.do02 AT %QX."X20CM8281g".DigitalOutput02;
	::io407Plus:cmModul12.ai01 AT %IW."X20CM8281g".AnalogInput01;
	::io407Plus:cmModul12.ao01 AT %QW."X20CM8281g".AnalogOutput01;
	::io407Plus:cmModul12.StatusInput01 AT %IB."X20CM8281g".StatusInput01;
	::io407Plus:cmModul13.di01 AT %IX."X20CM8281h".DigitalInput01;
	::io407Plus:cmModul13.di02 AT %IX."X20CM8281h".DigitalInput02;
	::io407Plus:cmModul13.di03 AT %IX."X20CM8281h".DigitalInput03;
	::io407Plus:cmModul13.di04 AT %IX."X20CM8281h".DigitalInput04;
	::io407Plus:cmModul13.do01 AT %QX."X20CM8281h".DigitalOutput01;
	::io407Plus:cmModul13.do02 AT %QX."X20CM8281h".DigitalOutput02;
	::io407Plus:cmModul13.ai01 AT %IW."X20CM8281h".AnalogInput01;
	::io407Plus:cmModul13.ao01 AT %QW."X20CM8281h".AnalogOutput01;
	::io407Plus:cmModul13.StatusInput01 AT %IB."X20CM8281h".StatusInput01;
	::io407Plus:cmModul14.di01 AT %IX."X20CM8281i".DigitalInput01;
	::io407Plus:cmModul14.di02 AT %IX."X20CM8281i".DigitalInput02;
	::io407Plus:cmModul14.di03 AT %IX."X20CM8281i".DigitalInput03;
	::io407Plus:cmModul14.di04 AT %IX."X20CM8281i".DigitalInput04;
	::io407Plus:cmModul14.do01 AT %QX."X20CM8281i".DigitalOutput01;
	::io407Plus:cmModul14.do02 AT %QX."X20CM8281i".DigitalOutput02;
	::io407Plus:cmModul14.ai01 AT %IW."X20CM8281i".AnalogInput01;
	::io407Plus:cmModul14.ao01 AT %QW."X20CM8281i".AnalogOutput01;
	::io407Plus:cmModul14.StatusInput01 AT %IB."X20CM8281i".StatusInput01;
	::io407Plus:cmModul15.di01 AT %IX."X20CM8281j".DigitalInput01;
	::io407Plus:cmModul15.di02 AT %IX."X20CM8281j".DigitalInput02;
	::io407Plus:cmModul15.di03 AT %IX."X20CM8281j".DigitalInput03;
	::io407Plus:cmModul15.di04 AT %IX."X20CM8281j".DigitalInput04;
	::io407Plus:cmModul15.do01 AT %QX."X20CM8281j".DigitalOutput01;
	::io407Plus:cmModul15.do02 AT %QX."X20CM8281j".DigitalOutput02;
	::io407Plus:cmModul15.ai01 AT %IW."X20CM8281j".AnalogInput01;
	::io407Plus:cmModul15.ao01 AT %QW."X20CM8281j".AnalogOutput01;
	::io407Plus:cmModul15.StatusInput01 AT %IB."X20CM8281j".StatusInput01;
	::Energiemes:apModulEnergie.PmeanT AT %IW."X20AP3131".PmeanT;
	::Energiemes:apModulEnergie.QmeanT AT %IW."X20AP3131".QmeanT;
	::Energiemes:apModulEnergie.SmeanT AT %IW."X20AP3131".SmeanT;
	::Energiemes:apModulEnergie.PFmeanT AT %IW."X20AP3131".PFmeanT;
	::Energiemes:apModulEnergie.AenergyT AT %ID."X20AP3131".AenergyT;
	::Energiemes:apModulEnergie.RenergyT AT %ID."X20AP3131".RenergyT;
	::Energiemes:apModulEnergie.SAenergyT AT %ID."X20AP3131".SAenergyT;
	::Energiemes:apModulEnergie.RBClearEnergy AT %IX."X20AP3131".RBClearEnergy;
	::Energiemes:apModulEnergie.TrigDFT AT %QX."X20AP3131".TrigDFT;
	::Energiemes:apModulEnergie.EnabEnergy AT %QX."X20AP3131".EnabEnergy;
	::Energiemes:apModulEnergie.ClearEnergy AT %QX."X20AP3131".ClearEnergy;
	::Energiemes:apModulEnergie.ForceEnergy AT %QX."X20AP3131".ForceEnergy;
	::io407Plus:diModul02.ModulOk AT %IX."X20DIF371".ModuleOk;
	::io407Plus:doModul03.ModulOk AT %IX."X20DO8322".ModuleOk;
	::io407Plus:brModul01.ModulOk AT %IX."X20BR7300".IF1.ST1.ModuleOk;
	::io407Plus:aiModul04.ModulOk AT %IX."X20AI8321".ModuleOk;
	::io407Plus:cmModul05.ModulOk AT %IX."X20CM8281".ModuleOk;
	::io407Plus:cmModul06.ModulOk AT %IX."X20CM8281a".ModuleOk;
	::io407Plus:cmModul07.ModulOk AT %IX."X20CM8281b".ModuleOk;
	::io407Plus:cmModul08.ModulOk AT %IX."X20CM8281c".ModuleOk;
	::io407Plus:cmModul09.ModulOk AT %IX."X20CM8281d".ModuleOk;
	::io407Plus:cmModul10.ModulOk AT %IX."X20CM8281e".ModuleOk;
	::io407Plus:cmModul11.ModulOk AT %IX."X20CM8281f".ModuleOk;
	::io407Plus:cmModul12.ModulOk AT %IX."X20CM8281g".ModuleOk;
	::io407Plus:cmModul13.ModulOk AT %IX."X20CM8281h".ModuleOk;
	::io407Plus:cmModul14.ModulOk AT %IX."X20CM8281i".ModuleOk;
	::io407Plus:cmModul15.ModulOk AT %IX."X20CM8281j".ModuleOk;
	::Energiemes:apModulEnergie.ModulOk AT %IX."X20AP3131".ModuleOk;
END_VAR
```

- Physical/4_07_Plus/4PPC30_0702_21B/PvMap.vvm: same as Physical/2_07/4PPC30_0702_21B/Cpu.per
- Physical/4_07_Plus/4PPC30_0702_21B/mappServices/Config.mprecipexml: same as Physical/2_07/4PPC30_0702_21B/mappServices/Config.mprecipexml
## Configuration HB3000_C30

CPU 4PPC30.0702-21B, AutomationRuntime C4.72, Build 4.1.2, Vc V4.72.0

### Task classes (Cpu.sw)
```
Cyclic#1 (cycle 10000 us, tolerance 10000 us):
  eUhr <- Util.eUhr.prg
  UsbLink <- CSV.UsbLink.prg
Cyclic#2 (cycle 20000 us, tolerance 20000 us):
  hmiMain <- Visualisierung.hmiMain.prg
  System <- Util.System.prg
  StartStopp <- Steuerung.StartStopp.prg
  mappPara <- Util.mappPara.prg
Cyclic#3 (cycle 50000 us, tolerance 50000 us):
  ioHB3000 <- IO.ioHB3000.prg
  aktorenMap <- IO.aktorenMapping.prg
  boxenMappi <- IO.boxenMapping.prg
  Ablaufstrg <- Ablaufsteuerung.Ablaufstrg.prg
  Leistung <- Regelung.Leistung.prg
  Sitemanage <- Sitemanager.Sitemanager.prg
Cyclic#4 (cycle 100000 us, tolerance 100000 us):
  Nutzung <- Util.Nutzung.prg
  Alarm <- Alarmsystem.Alarm.prg
  Berechnung <- Berechnung.Berechnung.prg
Cyclic#5 (cycle 200000 us, tolerance 200000 us):
  Energiemes <- IO.Energiemessung.prg
  hmiConnect <- Visualisierung.hmiConnect.prg
Cyclic#6 (cycle 500000 us, tolerance 500000 us):
  CSV01_EXT <- CSV.CSV01_EXT.prg
  CSV01_PRG <- CSV.CSV01_PRG.prg
DataObjects: CSV01_CFG <- CSV.CSV01_CFG.dob
VcDataObjects: Visu <- Visualisierung.Visu.dob
Libraries: operator, runtime, astime, AsIecCon, standard, sys_lib, AsBrStr, LascoMath, LascoReg, LascoTrock, LascoUtil, LaEntfV2, LascoBoxen, LoopConR, brsystem, asstring, FileIO, DataObj, AsARCfg, visapi, AsUSB, dvframe, IecCheck, AsTCP, MpFile, MpBase, MpRecipe, CControl, CSV
```

### Hardware
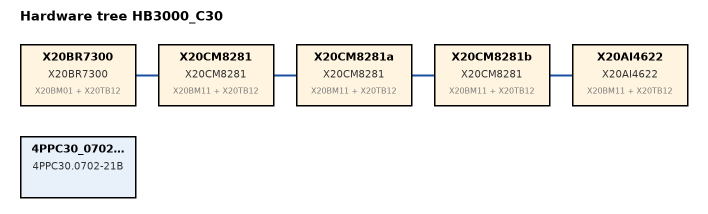
```
4PPC30_0702_21B : 4PPC30.0702-21B v1.1.4.0
  Connector IF3:
    ActivateDevice = 1
    Mode = Manual
    InternetAddress = 10.0.0.2
    SubnetMask = 255.255.255.0
    Vnc1
    VncVcObjectName1 = Visu
    VncKeyMappingFile1 = VC\PS2-Keyboard.dis
    VncMaxConnections1 = 5
    VncRefreshRate1 = 100
  Connector IF4:
    TerminatingResistor = 1
  ConfigurationID = CControl_HB3000_C30
  UserPartitionSize = 300
  RemanentGlobalPvSize = 6000
  EnableUsbRemoteInstall = 1
  TimerDeviceType = SWIOTIMER
  Cyclic1Duration = 10000
  Cyclic1Tolerance = 10000
  Cyclic2Duration = 20000
  Cyclic2Tolerance = 20000
  Cyclic3Duration = 50000
  Cyclic3Tolerance = 50000
  Cyclic4Duration = 100000
  Cyclic4Tolerance = 100000
  Cyclic5Duration = 200000
  Cyclic5Tolerance = 200000
  Cyclic6Duration = 500000
  Cyclic6Tolerance = 500000
  Cyclic7Duration = 1000000
  Cyclic7Tolerance = 1000000
  Cyclic8Duration = 10000
  Cyclic8Tolerance = 30000000
  FileDevice1
  FileDeviceName1 = CF
  FileDevicePath1 = F:\
  TimeZone = 140
  ActivateDaylightSavingTime = 1
  FtpUser1
  FtpUsername1 = lasco
  FtpUserPassword1 = Ef+S1okvKV7mfbBcr2vxnxcbPkrmnj/sE1vWqnyu2d8=
  FtpUserSalt1 = qtoxeAMd
  FTPAccessRight1 = 0
  FTPdevice1 = ALL
  VcObjectName = Visu
  KeyMappingFile = VC\4PPC30_0702_21B.dis
X20AI4622 : X20AI4622 v1.2.0.0  [SS1 -> X20TB12d.SS; SL -> X20BM11c.SL1]
  FunctionModel = CANIOBusController
  Supervision = off
  ChannelType01 = 4 to 20mA
  ChannelType02 = 4 to 20mA
X20BM01 : X20BM01 v2.2.0.0
X20BM11 : X20BM11 v1.1.0.0  [X2X1 -> X20BM01.IF1]
X20BM11a : X20BM11 v1.1.0.0  [X2X1 -> X20BM11.X2X2]
X20BM11b : X20BM11 v1.1.0.0  [X2X1 -> X20BM11a.X2X2]
X20BM11c : X20BM11 v1.1.0.0  [X2X1 -> X20BM11b.X2X2]
X20BR7300 : X20BR7300 v1.7.0.0  [CAN1 -> 4PPC30_0702_21B.IF4; SL -> X20BM01.SL1; SS1 -> X20TB12.SS]
  Supervision = off
X20CM8281 : X20CM8281 v1.4.0.0  [SS1 -> X20TB12a.SS; SL -> X20BM11.SL1]
  FunctionModel = CANIOBusController
  Supervision = off
  ChannelType01AI = 4 to 20mA
  LowerLimitAI = 0
  ChannelType01AO = 0 to 20mA
X20CM8281a : X20CM8281 v1.4.0.0  [SS1 -> X20TB12b.SS; SL -> X20BM11a.SL1]
  FunctionModel = CANIOBusController
  Supervision = off
  ChannelType01AI = 4 to 20mA
  LowerLimitAI = 0
  ChannelType01AO = 0 to 20mA
X20CM8281b : X20CM8281 v1.4.0.0  [SS1 -> X20TB12c.SS; SL -> X20BM11b.SL1]
  FunctionModel = CANIOBusController
  Supervision = off
  ChannelType01AI = 4 to 20mA
  LowerLimitAI = 0
  ChannelType01AO = 0 to 20mA
X20TB12 : X20TB12 v1.0.0.0
X20TB12a : X20TB12 v1.0.0.0
X20TB12b : X20TB12 v1.0.0.0
X20TB12c : X20TB12 v1.0.0.0
X20TB12d : X20TB12 v1.0.0.0
```

- Physical/HB3000_C30/4PPC30_0702_21B/Cpu.per: same as Physical/2_07/4PPC30_0702_21B/Cpu.per
### IoMap.iom - 4PPC30_0702_21B/IoMap.iom
```iecst
VAR_CONFIG
	::ioHB3000:brModul01.ModulOk AT %IX."X20BR7300".IF1.ST1.ModuleOk;
	::ioHB3000:cmModul02.ModulOk AT %IX."X20CM8281".ModuleOk;
	::ioHB3000:cmModul02.di01 AT %IX."X20CM8281".DigitalInput01;
	::ioHB3000:cmModul02.di02  AT %IX."X20CM8281".DigitalInput02;
	::ioHB3000:cmModul02.di03  AT %IX."X20CM8281".DigitalInput03;
	::ioHB3000:cmModul02.di04  AT %IX."X20CM8281".DigitalInput04;
	::ioHB3000:cmModul02.do01 AT %QX."X20CM8281".DigitalOutput01;
	::ioHB3000:cmModul02.do02 AT %QX."X20CM8281".DigitalOutput02;
	::ioHB3000:cmModul02.ai01 AT %IW."X20CM8281".AnalogInput01;
	::ioHB3000:cmModul02.ao01 AT %QW."X20CM8281".AnalogOutput01;
	::ioHB3000:cmModul02.StatusInput01 AT %IB."X20CM8281".StatusInput01;
	::ioHB3000:cmModul03.ModulOk AT %IX."X20CM8281a".ModuleOk;
	::ioHB3000:cmModul03.di01 AT %IX."X20CM8281a".DigitalInput01;
	::ioHB3000:cmModul03.di02 AT %IX."X20CM8281a".DigitalInput02;
	::ioHB3000:cmModul03.di03 AT %IX."X20CM8281a".DigitalInput03;
	::ioHB3000:cmModul03.di04 AT %IX."X20CM8281a".DigitalInput04;
	::ioHB3000:cmModul03.do01 AT %QX."X20CM8281a".DigitalOutput01;
	::ioHB3000:cmModul03.do02 AT %QX."X20CM8281a".DigitalOutput02;
	::ioHB3000:cmModul03.ai01 AT %IW."X20CM8281a".AnalogInput01;
	::ioHB3000:cmModul03.ao01 AT %QW."X20CM8281a".AnalogOutput01;
	::ioHB3000:cmModul03.StatusInput01 AT %IB."X20CM8281a".StatusInput01;
	::ioHB3000:cmModul04.ModulOk AT %IX."X20CM8281b".ModuleOk;
	::ioHB3000:cmModul04.di01 AT %IX."X20CM8281b".DigitalInput01;
	::ioHB3000:cmModul04.di02 AT %IX."X20CM8281b".DigitalInput02;
	::ioHB3000:cmModul04.di03 AT %IX."X20CM8281b".DigitalInput03;
	::ioHB3000:cmModul04.di04 AT %IX."X20CM8281b".DigitalInput04;
	::ioHB3000:cmModul04.do01 AT %QX."X20CM8281b".DigitalOutput01;
	::ioHB3000:cmModul04.do02 AT %QX."X20CM8281b".DigitalOutput02;
	::ioHB3000:cmModul04.ai01 AT %IW."X20CM8281b".AnalogInput01;
	::ioHB3000:cmModul04.ao01 AT %QW."X20CM8281b".AnalogOutput01;
	::ioHB3000:cmModul04.StatusInput01 AT %IB."X20CM8281b".StatusInput01;
	::ioHB3000:aiModul05.ModulOk AT %IX."X20AI4622".ModuleOk;
	::ioHB3000:aiModul05.ai01 AT %IW."X20AI4622".AnalogInput01;
	::ioHB3000:aiModul05.ai02 AT %IW."X20AI4622".AnalogInput02;
	::ioHB3000:aiModul05.ai03 AT %IW."X20AI4622".AnalogInput03;
	::ioHB3000:aiModul05.ai04 AT %IW."X20AI4622".AnalogInput04;
	::ioHB3000:aiModul05.StatusInput01 AT %IB."X20AI4622".StatusInput01;
END_VAR
```

- Physical/HB3000_C30/4PPC30_0702_21B/PvMap.vvm: same as Physical/2_07/4PPC30_0702_21B/Cpu.per
- Physical/HB3000_C30/4PPC30_0702_21B/mappServices/Config.mprecipexml: same as Physical/2_07/4PPC30_0702_21B/mappServices/Config.mprecipexml
## Configuration HB4000_C30

CPU 4PPC30.0702-21B, AutomationRuntime C4.72, Build 4.1.2, Vc V4.72.0

### Task classes (Cpu.sw)
```
Cyclic#1 (cycle 10000 us, tolerance 10000 us):
  eUhr <- Util.eUhr.prg
  UsbLink <- CSV.UsbLink.prg
Cyclic#2 (cycle 20000 us, tolerance 20000 us):
  hmiMain <- Visualisierung.hmiMain.prg
  System <- Util.System.prg
  StartStopp <- Steuerung.StartStopp.prg
  mappPara <- Util.mappPara.prg
Cyclic#3 (cycle 50000 us, tolerance 50000 us):
  ioHB4000 <- IO.ioHB4000.prg
  aktorenMap <- IO.aktorenMapping.prg
  boxenMappi <- IO.boxenMapping.prg
  Ablaufstrg <- Ablaufsteuerung.Ablaufstrg.prg
  Leistung <- Regelung.Leistung.prg
  Sitemanage <- Sitemanager.Sitemanager.prg
Cyclic#4 (cycle 100000 us, tolerance 100000 us):
  Nutzung <- Util.Nutzung.prg
  Alarm <- Alarmsystem.Alarm.prg
  Berechnung <- Berechnung.Berechnung.prg
Cyclic#5 (cycle 200000 us, tolerance 200000 us):
  Energiemes <- IO.Energiemessung.prg
  hmiConnect <- Visualisierung.hmiConnect.prg
Cyclic#6 (cycle 500000 us, tolerance 500000 us):
  CSV01_EXT <- CSV.CSV01_EXT.prg
  CSV01_PRG <- CSV.CSV01_PRG.prg
DataObjects: CSV01_CFG <- CSV.CSV01_CFG.dob
VcDataObjects: Visu <- Visualisierung.Visu.dob
Libraries: CControl, operator, runtime, astime, AsIecCon, standard, sys_lib, AsBrStr, LascoMath, LascoReg, LascoTrock, LascoUtil, LaEntfV2, LascoBoxen, LoopConR, brsystem, asstring, FileIO, DataObj, AsARCfg, visapi, AsUSB, dvframe, IecCheck, AsTCP, MpFile, MpBase, MpRecipe, CSV
```

### Hardware
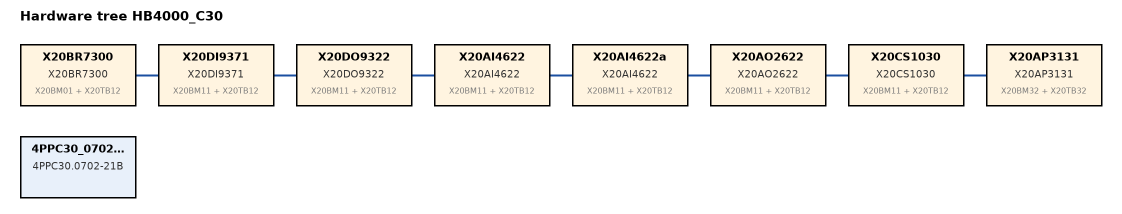
```
4PPC30_0702_21B : 4PPC30.0702-21B v1.1.4.0
  Connector IF3:
    ActivateDevice = 1
    Mode = Manual
    InternetAddress = 10.0.0.2
    SubnetMask = 255.255.255.0
    Vnc1
    VncVcObjectName1 = Visu
    VncKeyMappingFile1 = VC\PS2-Keyboard.dis
    VncMaxConnections1 = 5
    VncRefreshRate1 = 100
  Connector IF4:
    TerminatingResistor = 1
  ConfigurationID = CControl_HB4000_C30
  UserPartitionSize = 300
  RemanentGlobalPvSize = 6000
  EnableUsbRemoteInstall = 1
  TimerDeviceType = SWIOTIMER
  Cyclic1Duration = 10000
  Cyclic1Tolerance = 10000
  Cyclic2Duration = 20000
  Cyclic2Tolerance = 20000
  Cyclic3Duration = 50000
  Cyclic3Tolerance = 50000
  Cyclic4Duration = 100000
  Cyclic4Tolerance = 100000
  Cyclic5Duration = 200000
  Cyclic5Tolerance = 200000
  Cyclic6Duration = 500000
  Cyclic6Tolerance = 500000
  Cyclic7Duration = 1000000
  Cyclic7Tolerance = 1000000
  Cyclic8Duration = 10000
  Cyclic8Tolerance = 30000000
  FileDevice1
  FileDeviceName1 = CF
  FileDevicePath1 = F:\
  TimeZone = 140
  ActivateDaylightSavingTime = 1
  FtpUser1
  FtpUsername1 = lasco
  FtpUserPassword1 = sI+AZni0GkarZ1kwqy/tAOF5J+WJqiGmH88ZxWXRWSc=
  FtpUserSalt1 = SrIaQtpG
  FTPAccessRight1 = 0
  FTPdevice1 = ALL
  VcObjectName = Visu
  KeyMappingFile = VC\4PPC30_0702_21B.dis
X20AI4622 : X20AI4622 v1.2.0.0  [SS1 -> X20TB12c.SS; SL -> X20BM11b.SL1]
  FunctionModel = CANIOBusController
  Supervision = off
  LowerLimit = 0
  ChannelType01 = 4 to 20mA
  ChannelType02 = 4 to 20mA
  ChannelType03 = 4 to 20mA
  ChannelType04 = 4 to 20mA
X20AI4622a : X20AI4622 v1.2.0.0  [SS1 -> X20TB12d.SS; SL -> X20BM11c.SL1]
  FunctionModel = CANIOBusController
  Supervision = off
  ChannelType01 = 4 to 20mA
  ChannelType02 = 4 to 20mA
  ChannelType03 = 4 to 20mA
X20AO2622 : X20AO2622 v1.3.0.0  [SS1 -> X20TB12e.SS; SL -> X20BM11d.SL1]
  FunctionModel = CANIOBusController
  Supervision = off
  ChannelType01 = 0 to 20mA
  ChannelType02 = 0 to 20mA
X20AP3131 : X20AP3131 v1.5.0.0  [SS1 -> X20TB32.SS; SL -> X20BM32.SL1]
  FunctionModel = CANIOBusController
  Supervision = off
  CurrentRatioA = 50
  CurrentRatioB = 50
  CurrentRatioC = 50
X20BM01 : X20BM01 v2.2.0.0
X20BM11 : X20BM11 v1.1.0.0  [X2X1 -> X20BM01.IF1]
X20BM11a : X20BM11 v1.1.0.0  [X2X1 -> X20BM11.X2X2]
X20BM11b : X20BM11 v1.1.0.0  [X2X1 -> X20BM11a.X2X2]
X20BM11c : X20BM11 v1.1.0.0  [X2X1 -> X20BM11b.X2X2]
X20BM11d : X20BM11 v1.1.0.0  [X2X1 -> X20BM11c.X2X2]
X20BM11e : X20BM11 v1.1.0.0  [X2X1 -> X20BM11d.X2X2]
X20BM32 : X20BM32 v1.1.0.0  [X2X1 -> X20BM11e.X2X2]
X20BR7300 : X20BR7300 v1.7.0.0  [CAN1 -> 4PPC30_0702_21B.IF4; SL -> X20BM01.SL1; SS1 -> X20TB12.SS]
  Supervision = off
X20CS1030 : X20CS1030 v1.8.0.0  [SS1 -> X20TB12f.SS; SL -> X20BM11e.SL1]
  FunctionModel = CANIOBusController
  Supervision = off
X20DI9371 : X20DI9371 v1.4.0.0  [SS1 -> X20TB12a.SS; SL -> X20BM11.SL1]
  FunctionModel = CANIOBusController
  Supervision = off
X20DO9322 : X20DO9322 v1.7.0.0  [SS1 -> X20TB12b.SS; SL -> X20BM11a.SL1]
  FunctionModel = CANIOBusController
  Supervision = off
X20TB12 : X20TB12 v1.0.0.0
X20TB12a : X20TB12 v1.0.0.0
X20TB12b : X20TB12 v1.0.0.0
X20TB12c : X20TB12 v1.0.0.0
X20TB12d : X20TB12 v1.0.0.0
X20TB12e : X20TB12 v1.0.0.0
X20TB12f : X20TB12 v1.0.0.0
X20TB32 : X20TB32 v1.0.0.1
```

- Physical/HB4000_C30/4PPC30_0702_21B/Cpu.per: same as Physical/2_07/4PPC30_0702_21B/Cpu.per
### IoMap.iom - 4PPC30_0702_21B/IoMap.iom
```iecst
VAR_CONFIG
	::ioHB4000:brModul01.ModulOk AT %IX."X20BR7300".IF1.ST1.ModuleOk;
	::ioHB4000:diModul02.ModulOk AT %IX."X20DI9371".ModuleOk;
	::ioHB4000:diModul02.di01 AT %IX."X20DI9371".DigitalInput01;
	::ioHB4000:diModul02.di02  AT %IX."X20DI9371".DigitalInput02;
	::ioHB4000:diModul02.di03  AT %IX."X20DI9371".DigitalInput03;
	::ioHB4000:diModul02.di04  AT %IX."X20DI9371".DigitalInput04;
	::ioHB4000:diModul02.di05  AT %IX."X20DI9371".DigitalInput05;
	::ioHB4000:diModul02.di06  AT %IX."X20DI9371".DigitalInput06;
	::ioHB4000:diModul02.di07  AT %IX."X20DI9371".DigitalInput07;
	::ioHB4000:diModul02.di08  AT %IX."X20DI9371".DigitalInput08;
	::ioHB4000:diModul02.di09  AT %IX."X20DI9371".DigitalInput09;
	::ioHB4000:diModul02.di10  AT %IX."X20DI9371".DigitalInput10;
	::ioHB4000:diModul02.di11  AT %IX."X20DI9371".DigitalInput11;
	::ioHB4000:diModul02.di12  AT %IX."X20DI9371".DigitalInput12;
	::ioHB4000:doModul03.ModulOk AT %IX."X20DO9322".ModuleOk;
	::ioHB4000:doModul03.do01 AT %QX."X20DO9322".DigitalOutput01;
	::ioHB4000:doModul03.do02  AT %QX."X20DO9322".DigitalOutput02;
	::ioHB4000:doModul03.do03  AT %QX."X20DO9322".DigitalOutput03;
	::ioHB4000:doModul03.do04  AT %QX."X20DO9322".DigitalOutput04;
	::ioHB4000:doModul03.do05  AT %QX."X20DO9322".DigitalOutput05;
	::ioHB4000:doModul03.do06  AT %QX."X20DO9322".DigitalOutput06;
	::ioHB4000:doModul03.do07  AT %QX."X20DO9322".DigitalOutput07;
	::ioHB4000:doModul03.do08  AT %QX."X20DO9322".DigitalOutput08;
	::ioHB4000:doModul03.do09  AT %QX."X20DO9322".DigitalOutput09;
	::ioHB4000:doModul03.do10  AT %QX."X20DO9322".DigitalOutput10;
	::ioHB4000:doModul03.do11  AT %QX."X20DO9322".DigitalOutput11;
	::ioHB4000:doModul03.do12  AT %QX."X20DO9322".DigitalOutput12;
	::ioHB4000:aiModul04.ModulOk AT %IX."X20AI4622".ModuleOk;
	::ioHB4000:aiModul04.ai01 AT %IW."X20AI4622".AnalogInput01;
	::ioHB4000:aiModul04.ai02 AT %IW."X20AI4622".AnalogInput02;
	::ioHB4000:aiModul04.ai03 AT %IW."X20AI4622".AnalogInput03;
	::ioHB4000:aiModul04.ai04 AT %IW."X20AI4622".AnalogInput04;
	::ioHB4000:aiModul04.StatusInput01 AT %IB."X20AI4622".StatusInput01;
	::ioHB4000:aiModul05.ModulOk AT %IX."X20AI4622a".ModuleOk;
	::ioHB4000:aiModul05.ai01 AT %IW."X20AI4622a".AnalogInput01;
	::ioHB4000:aiModul05.ai02 AT %IW."X20AI4622a".AnalogInput02;
	::ioHB4000:aiModul05.ai03 AT %IW."X20AI4622a".AnalogInput03;
	::ioHB4000:aiModul05.ai04 AT %IW."X20AI4622a".AnalogInput04;
	::ioHB4000:aiModul05.StatusInput01 AT %IB."X20AI4622a".StatusInput01;
	::ioHB4000:aoModul06.ModulOk AT %IX."X20AO2622".ModuleOk;
	::ioHB4000:aoModul06.ao01 AT %QW."X20AO2622".AnalogOutput01;
	::ioHB4000:aoModul06.ao02 AT %QW."X20AO2622".AnalogOutput02;
	::ioHB4000:csModul07 AT %IX."X20CS1030".ModuleOk;
	::Energiemes:apModulEnergie.ModulOk AT %IX."X20AP3131".ModuleOk;
	::Energiemes:apModulEnergie.PmeanT AT %IW."X20AP3131".PmeanT;
	::Energiemes:apModulEnergie.QmeanT AT %IW."X20AP3131".QmeanT;
	::Energiemes:apModulEnergie.SmeanT AT %IW."X20AP3131".SmeanT;
	::Energiemes:apModulEnergie.PFmeanT AT %IW."X20AP3131".PFmeanT;
	::Energiemes:apModulEnergie.AenergyT AT %ID."X20AP3131".AenergyT;
	::Energiemes:apModulEnergie.RenergyT AT %ID."X20AP3131".RenergyT;
	::Energiemes:apModulEnergie.SAenergyT AT %ID."X20AP3131".SAenergyT;
	::Energiemes:apModulEnergie.RBClearEnergy AT %IX."X20AP3131".RBClearEnergy;
	::Energiemes:apModulEnergie.TrigDFT AT %QX."X20AP3131".TrigDFT;
	::Energiemes:apModulEnergie.EnabEnergy AT %QX."X20AP3131".EnabEnergy;
	::Energiemes:apModulEnergie.ClearEnergy AT %QX."X20AP3131".ClearEnergy;
	::Energiemes:apModulEnergie.ForceEnergy AT %QX."X20AP3131".ForceEnergy;
END_VAR
```

- Physical/HB4000_C30/4PPC30_0702_21B/PvMap.vvm: same as Physical/2_07/4PPC30_0702_21B/Cpu.per
- Physical/HB4000_C30/4PPC30_0702_21B/mappServices/Config.mprecipexml: same as Physical/2_07/4PPC30_0702_21B/mappServices/Config.mprecipexml
## Configuration Sim

CPU PC_any, AutomationRuntime F4.73, Build 4.1.2, Vc V4.72.6

### Task classes (Cpu.sw)
```
Cyclic#1 (cycle 20000 us):
  eUhr <- Util.eUhr.prg
  mappPara <- Util.mappPara.prg
  hmiMain <- Visualisierung.hmiMain.prg
Cyclic#2 (cycle 50000 us):
  StartStopp <- Steuerung.StartStopp.prg
  Berechnung <- Berechnung.Berechnung.prg
  aktorenMap <- IO.aktorenMapping.prg
  boxenMappi <- IO.boxenMapping.prg
  Alarm <- Alarmsystem.Alarm.prg
  Ablaufstrg <- Ablaufsteuerung.Ablaufstrg.prg
  Leistung <- Regelung.Leistung.prg
  hmiConnect <- Visualisierung.hmiConnect.prg
Cyclic#3:
  Nutzung <- Util.Nutzung.prg
VcDataObjects: Visu <- Visualisierung.Visu.dob
Binaries: vcpkat, vccdt, vccbmp, Visu03, vcfile, arial, vctcal, vcrt, vcmgr, arsvcreg, vccstr, vcbclass, vccbtn, vcgclass, vcdsint, vcnet, vccline, vcshared, vcclbox, vccddbox, arialbd, vccnum, vcpdvnc, FWRules, vccalarm, visvc, vcpfar00, vccbar, vcctext, Visu01, vcpdsw, vcfntttf, vccovl, vccshape, vcalarm, Visu02, vcctrend, udbdef, vccpopup, vcdsloc, vcchspot, TCData, arconfig, asfw, iomap, Role, ashwd, Config, ashwac, sysconf, User
Libraries: operator, runtime, astime, AsIecCon, standard, sys_lib, AsBrStr, LascoMath, LascoReg, LascoTrock, LascoUtil, LaEntfV2, LascoBoxen, LoopConR, brsystem, asstring, FileIO, DataObj, AsARCfg, visapi, AsUSB, dvframe, IecCheck, AsTCP, MpRecipe, MpBase, MpFile, vcresman
```

### Hardware
```
PC : PC_any v1.1.1.0 (OrderNumber=PC)
  Connector IF3:
    Vnc1
    VncVcObjectName1 = Visu
    VncKeyMappingFile1 = VC\PS2-Keyboard2.dis
    VncRefreshRate1 = 100
  ConfigurationID = LaTronicCcontrolPlus407_Test
  RemanentGlobalPvSize = 5000
  Cyclic1Duration = 20000
  Cyclic2Duration = 50000
  FileDevice1
  FileDeviceName1 = CF
  FileDevicePath1 = C:\Users\rlachner\Documents\mappParameter
  FtpUser1
  FtpUsername1 = lasco
  FtpUserPassword1 = XXwjkhGq37/etuSmmp0wfzbic2StEj7ZqLjdnjOpFzU=
  FtpUserSalt1 = ZwaEHSD6
  FTPAccessRight1 = 0
  FTPdevice1 = ALL
```

- Physical/Sim/PC/Cpu.per: same as Physical/2_07/4PPC30_0702_21B/Cpu.per
- Physical/Sim/PC/IoMap.iom: same as Physical/2_07/4PPC30_0702_21B/Cpu.per
- Physical/Sim/PC/PvMap.vvm: same as Physical/2_07/4PPC30_0702_21B/Cpu.per
- Physical/Sim/PC/mappServices/Config.mprecipexml: same as Physical/2_07/4PPC30_0702_21B/mappServices/Config.mprecipexml
## Logical view

Binary libraries used (declarations not repeated): operator, runtime, astime, AsIecCon, standard, sys_lib, AsBrStr, LoopConR 4.10.0, brsystem, asstring, FileIO, DataObj, AsARCfg, visapi, AsUSB, dvframe, AsTCP, MpBase 5.24.1, MpFile 5.24.6, MpRecipe 5.24.6
